# B&R Automation Studio project NAELD004C00R10L518F00 (part 16)

#### Act_OptP0950Ctrl.st
```iecst
ACTION Act_OptP0950Ctrl:

////Control
//	IF g_tyP0950Simu.tySimu.tyHotspotSimu.bRtCompl = TRUE THEN
//		g_tyP0950Simu.tySimu.tyHotspotSimu.bRtCompl	:= FALSE;
//
//		fUIInRtStatOff(ADR(g_tyP0950Simu.tySimuCtrl.tyLyr.uiRtStat));
//	END_IF
//
//	IF g_tyP0950Simu.tySimuCtrl.tyLyr.uiRtStat.0 = FALSE THEN
//		IF g_tyP0950Simu.tySimuCtrl.tyBtnStart.bRtCompl = TRUE THEN
//			g_tyP0950Simu.tySimuCtrl.tyBtnStart.bRtComplm	:= FALSE;
//
//			IF tyOpsProgData.bSimuCycStpCtrl = TRUE THEN
//				tyOpsProgData.bSimuCycStpCtrl	:= FALSE;
//			END_IF
//
//			IF tyOpsProgData.bAutoStepCtrl = TRUE THEN
//				tyOpsProgData.bAutoStepCtrl	:= FALSE;
//			END_IF
//
//			tyOpsProgData.bSimuCtrl	:= TRUE;
//			fUIInRtStatHide(ADR(g_tyP0950Simu.tySimuCtrl.tyLyr.uiRtStat));
//
//		ELSIF g_tyP0950Simu.tySimuCtrl.tyBtnStop.bRtCompl = TRUE THEN
//			g_tyP0950Simu.tySimuCtrl.tyBtnStop.bRtCompl	:= FALSE;
//
//			tyOpsProgData.bSimuCycStpCtrl	:= TRUE;
//			fUIInRtStatHide(ADR(g_tyP0950Simu.tySimuCtrl.tyLyr.uiRtStat));
//
//		ELSIF g_tyP0950Simu.tySimuCtrl.tyBtnStep.bRtCompl = TRUE THEN
//			g_tyP0950Simu.tySimuCtrl.tyBtnStep.bRtCompl	:= FALSE;
//
//			IF tyOpsProgData.bAutoStepCtrl = FALSE THEN
//				tyOpsProgData.bSimuCtrl			:= TRUE;
//				tyOpsProgData.bAutoStepCtrl		:= TRUE;
//				tyOpsProgData.bSimuCycStpCtrl	:= FALSE;
//			ELSIF tyOpsProgData.bSimuCycStpCtrl = TRUE THEN
//				tyOpsProgData.bSimuCycStpCtrl	:= FALSE;
//			ELSE
//				tyOpsProgData.bAutoStepRunCtrl	:= TRUE;
//			END_IF
//		ELSIF g_tyP0950Simu.tySimuCtrl.tyHotspotClose.bRtCompl = TRUE THEN
//			g_tyP0950Simu.tySimuCtrl.tyHotspotClose.bRtCompl	:= FALSE;
//
//			fUIInRtStatHide(ADR(g_tyP0950Simu.tySimuCtrl.tyLyr.uiRtStat));
//		END_IF
//	END_IF
//
//	//Display
//	IF tyOpsProgData.bSimuCtrl = TRUE AND tyOpsProgData.bSimuCycStpCtrl = TRUE THEN
//		fUIInRtStatOff(ADR(g_tyP0950Simu.tySimu.tyBtnStartStat.uiRtStat));
//		fUIInRtStatHide(ADR(g_tyP0950Simu.tySimu.tyBtnStopStat.uiRtStat));
//		fUIInRtStatHide(ADR(g_tyP0950Simu.tySimu.tyBtnStepStat.uiRtStat));
//
//		fbStopBlinkTm(IN := TRUE);
//		IF fbStopBlinkTm.Q = TRUE THEN
//			fbStopBlinkTm(IN := FALSE);
//
//			g_tyP0950Simu.tySimu.tyBtnStartStat.bValue	:= NOT g_tyP0950Simu.tySimu.tyBtnStartStat.bValue;
//		END_IF
//	ELSIF tyOpsProgData.bSimuCtrl = TRUE AND tyOpsProgData.bAutoStepCtrl = TRUE THEN
//		fUIInRtStatHide(ADR(g_tyP0950Simu.tySimu.tyBtnStartStat.uiRtStat));
//		fUIInRtStatHide(ADR(g_tyP0950Simu.tySimu.tyBtnStopStat.uiRtStat));
//		fUIInRtStatOff(ADR(g_tyP0950Simu.tySimu.tyBtnStepStat.uiRtStat));
//	ELSIF tyOpsProgData.bSimuCtrl = TRUE THEN
//		fUIInRtStatOff(ADR(g_tyP0950Simu.tySimu.tyBtnStartStat.uiRtStat));
//		fUIInRtStatHide(ADR(g_tyP0950Simu.tySimu.tyBtnStopStat.uiRtStat));
//		fUIInRtStatHide(ADR(g_tyP0950Simu.tySimu.tyBtnStepStat.uiRtStat));
//
//		g_tyP0950Simu.tySimu.tyBtnStartStat.bValue	:= FALSE;
//	ELSE
//		fUIInRtStatHide(ADR(g_tyP0950Simu.tySimu.tyBtnStartStat.uiRtStat));
//		fUIInRtStatOff(ADR(g_tyP0950Simu.tySimu.tyBtnStopStat.uiRtStat));
//		fUIInRtStatHide(ADR(g_tyP0950Simu.tySimu.tyBtnStepStat.uiRtStat));
//	END_IF
//
//	//Mask
//	IF bErr = TRUE THEN
//		fUIInRtStatOff(ADR(g_tyP0950Simu.tySimu.tyHotspotSimu.uiMaskRtStat));
//	ELSE
//		fUIInRtStatHide(ADR(g_tyP0950Simu.tySimu.tyHotspotSimu.uiMaskRtStat));
//	END_IF

	// Error
	IF EDGEPOS(p_bAlarmErr = TRUE AND p_bSimuStatusStop = FALSE) THEN

		tyP0950Simu.tySimu.tyBtnStart.bRtCompl	:= FALSE;
		tyP0950Simu.tySimu.tyBtnStop.bRtCompl	:= FALSE;
		tyP0950Simu.tySimu.tyBtnInShutterSim.bRtCompl	:= FALSE;

		tyP0950Simu.tySimu.tyBtnStart.bValue	:= FALSE;
		tyP0950Simu.tySimu.tyBtnStop.bValue		:= FALSE;
		tyP0950Simu.tySimu.tyBtnInShutterSim.bValue	:= FALSE;

		eSimuAct	:= SimulationsActError;

	ELSE

		IF p_eSimuStat = SimulationsActError AND p_eSimuStatus = Done THEN
			eSimuAct	:= SimulationsActIdle;

		END_IF

	END_IF

	//Control
	IF tyP0950Simu.tySimu.tyBtnStart.bRtCompl = TRUE THEN
		tyP0950Simu.tySimu.tyBtnStop.bRtCompl	:= FALSE;

		eSimuAct		:= SimulationsActStart;

		IF p_eSimuStat = SimulationsActStart AND p_eSimuStatus = Done THEN
			eSimuAct	:= SimulationsActIdle;

			tyP0950Simu.tySimu.tyBtnStart.bRtCompl	:= FALSE;

		END_IF

	ELSIF tyP0950Simu.tySimu.tyBtnStop.bRtCompl = TRUE THEN
		tyP0950Simu.tySimu.tyBtnStart.bRtCompl	:= FALSE;

		eSimuAct			:= SimulationsActStop;

		IF p_eSimuStat = SimulationsActStop AND p_eSimuStatus = Done THEN
			eSimuAct		:= SimulationsActIdle;

			tyP0950Simu.tySimu.tyBtnStop.bRtCompl	:= FALSE;
		END_IF

	END_IF

	// Mask
	IF p_bAlarmErr = TRUE OR (p_tyDI.bSafetyRlySig = FALSE) THEN
		fUIInRtStatOff(ADR(tyP0950Simu.tySimu.tyBtnStart.uiMaskRtStat));
		fUIInRtStatOff(ADR(tyP0950Simu.tySimu.tyBtnStop.uiMaskRtStat));

	ELSIF p_bSimuStatusCycleStop = TRUE THEN
		fUIInRtStatHide(ADR(tyP0950Simu.tySimu.tyBtnStart.uiMaskRtStat));
		fUIInRtStatOff(ADR(tyP0950Simu.tySimu.tyBtnStop.uiMaskRtStat));

		fbStopBlinkTm(IN := TRUE);
		IF fbStopBlinkTm.Q = TRUE THEN
			fbStopBlinkTm(IN := FALSE);

			tyP0950Simu.tySimu.tyBtnStart.bValue		:= NOT tyP0950Simu.tySimu.tyBtnStart.bValue;
		END_IF

	ELSIF p_bSimuStatusRun = TRUE THEN
		fUIInRtStatOff(ADR(tyP0950Simu.tySimu.tyBtnStart.uiMaskRtStat));
		fUIInRtStatHide(ADR(tyP0950Simu.tySimu.tyBtnStop.uiMaskRtStat));

	ELSE
		fUIInRtStatHide(ADR(tyP0950Simu.tySimu.tyBtnStart.uiMaskRtStat));
		fUIInRtStatOff(ADR(tyP0950Simu.tySimu.tyBtnStop.uiMaskRtStat));

	END_IF

	//AGV Simulatiom
	IF tyP0950Simu.tyAGVToMc.tyBtnAGVSimulateOn.bRtCompl THEN
		IF tyP0950Simu.tyAGVToMc.tyBtnAGVSimulateOn.bValue THEN
			bAGVSimulationOn	:= TRUE;
			tyP0950Simu.tyAGVToMc.tyBtnAGVSimulateOn.bRtCompl:= FALSE;
		ELSE
			bAGVSimulationOn := FALSE;
			tyP0950Simu.tyAGVToMc.tyBtnAGVSimulateOn.bRtCompl:= FALSE;
		END_IF
	END_IF

	IF tyP0950Simu.tyAGVToMc.tyBtnAGVOnline.bRtCompl THEN
		IF tyP0950Simu.tyAGVToMc.tyBtnAGVOnline.bValue THEN
			bAGVSimulateOnline := TRUE;
			tyP0950Simu.tyAGVToMc.tyBtnAGVOnline.bRtCompl := FALSE;
		ELSE
			bAGVSimulateOnline := FALSE;
			tyP0950Simu.tyAGVToMc.tyBtnAGVOnline.bRtCompl := FALSE;
		END_IF
	END_IF

	IF tyP0950Simu.tyAGVToMc.tyBtnAGVAuto.bRtCompl THEN
		IF tyP0950Simu.tyAGVToMc.tyBtnAGVAuto.bValue THEN
			tyAGVSimulateSig.bVEHAuto := TRUE;
			tyP0950Simu.tyAGVToMc.tyBtnAGVAuto.bRtCompl:= FALSE;
		ELSE
			tyAGVSimulateSig.bVEHAuto := FALSE;
			tyP0950Simu.tyAGVToMc.tyBtnAGVAuto.bRtCompl:= FALSE;
		END_IF
	END_IF

	IF tyP0950Simu.tyAGVToMc.tyBtnAGVInPos1.bRtCompl THEN
		IF tyP0950Simu.tyAGVToMc.tyBtnAGVInPos1.bValue THEN
			tyAGVSimulateSig.bVEHInPos1 := TRUE;
			tyP0950Simu.tyAGVToMc.tyBtnAGVInPos1.bRtCompl:= FALSE;
		ELSE
			tyAGVSimulateSig.bVEHInPos1 := FALSE;
			tyP0950Simu.tyAGVToMc.tyBtnAGVInPos1.bRtCompl:= FALSE;
		END_IF
	END_IF

	IF tyP0950Simu.tyAGVToMc.tyBtnAGVInPos2.bRtCompl THEN
		IF tyP0950Simu.tyAGVToMc.tyBtnAGVInPos2.bValue THEN
			tyAGVSimulateSig.bVEHInPos2 := TRUE;
			tyP0950Simu.tyAGVToMc.tyBtnAGVInPos2.bRtCompl:= FALSE;
		ELSE
			tyAGVSimulateSig.bVEHInPos2 := FALSE;
			tyP0950Simu.tyAGVToMc.tyBtnAGVInPos2.bRtCompl:= FALSE;
		END_IF
	END_IF

	IF tyP0950Simu.tyAGVToMc.tyBtnAGVInPos3.bRtCompl THEN
		IF tyP0950Simu.tyAGVToMc.tyBtnAGVInPos3.bValue THEN
			tyAGVSimulateSig.bVEHInPos3 := TRUE;
			tyP0950Simu.tyAGVToMc.tyBtnAGVInPos3.bRtCompl:= FALSE;
		ELSE
			tyAGVSimulateSig.bVEHInPos3 := FALSE;
			tyP0950Simu.tyAGVToMc.tyBtnAGVInPos3.bRtCompl:= FALSE;
		END_IF
	END_IF

	IF tyP0950Simu.tyAGVToMc.tyBtnAGV1Occupied.bRtCompl THEN
		IF tyP0950Simu.tyAGVToMc.tyBtnAGV1Occupied.bValue THEN
			tyAGVSimulateSig.bVEH1Occupied := TRUE;
			tyP0950Simu.tyAGVToMc.tyBtnAGV1Occupied.bRtCompl := FALSE;
		ELSE
			tyAGVSimulateSig.bVEH1Occupied := FALSE;
			tyP0950Simu.tyAGVToMc.tyBtnAGV1Occupied.bRtCompl := FALSE;
		END_IF
	END_IF

	IF tyP0950Simu.tyAGVToMc.tyBtnAGV2Occupied.bRtCompl THEN
		IF tyP0950Simu.tyAGVToMc.tyBtnAGV2Occupied.bValue THEN
			tyAGVSimulateSig.bVEH2Occupied := TRUE;
			tyP0950Simu.tyAGVToMc.tyBtnAGV2Occupied.bRtCompl := FALSE;
		ELSE
			tyAGVSimulateSig.bVEH2Occupied := FALSE;
			tyP0950Simu.tyAGVToMc.tyBtnAGV2Occupied.bRtCompl := FALSE;
		END_IF
	END_IF

	IF tyP0950Simu.tyAGVToMc.tyBtnAGV3Occupied.bRtCompl THEN
		IF tyP0950Simu.tyAGVToMc.tyBtnAGV3Occupied.bValue THEN
			tyAGVSimulateSig.bVEH3Occupied := TRUE;
			tyP0950Simu.tyAGVToMc.tyBtnAGV3Occupied.bRtCompl := FALSE;
		ELSE
			tyAGVSimulateSig.bVEH3Occupied := FALSE;
			tyP0950Simu.tyAGVToMc.tyBtnAGV3Occupied.bRtCompl := FALSE;
		END_IF
	END_IF

	//Machine to AGV Communication
	tyP0950Simu.tyMcToAGV.tyBtnMachineOnline.bValue := p_bMachineOnline;
	tyP0950Simu.tyMcToAGV.tyBtnMachineEstop.bValue	:= p_tyDTMagToAGV.bEStopErr;

	//Magazine #1 to AGV Communication
	tyP0950Simu.tyMcToAGV.tyBtnMag1Auto.bValue				:= p_tyDTMagToAGV.bCI1Auto;
	tyP0950Simu.tyMcToAGV.tyBtnMag1Empty.bValue				:= p_tyDTMagToAGV.bCI1MagazineEmpty;
	tyP0950Simu.tyMcToAGV.tyBtnMag1IncorrectModel.bValue	:= p_tyDTMagToAGV.bCI1IncorrectMagazineModel;
	tyP0950Simu.tyMcToAGV.tyBtnMag1Occupied.bValue			:= p_tyDTMagToAGV.bCI1Occupied;
	tyP0950Simu.tyMcToAGV.tyBtnMag1Rdy.bValue				:= p_tyDTMagToAGV.bCI1Rdy;

	//Magazine #2 to AGV Communication
	tyP0950Simu.tyMcToAGV.tyBtnMag2Auto.bValue				:= p_tyDTMagToAGV.bCI2Auto;
	tyP0950Simu.tyMcToAGV.tyBtnMag2Empty.bValue				:= p_tyDTMagToAGV.bCI2MagazineEmpty;
	tyP0950Simu.tyMcToAGV.tyBtnMag2IncorrectModel.bValue	:= p_tyDTMagToAGV.bCI2IncorrectMagazineModel;
	tyP0950Simu.tyMcToAGV.tyBtnMag2Occupied.bValue			:= p_tyDTMagToAGV.bCI2Occupied;
	tyP0950Simu.tyMcToAGV.tyBtnMag2Rdy.bValue				:= p_tyDTMagToAGV.bCI2Rdy;

	//Magazine #3 to AGV Communication
	tyP0950Simu.tyMcToAGV.tyBtnMag3Auto.bValue				:= p_tyDTMagToAGV.bCI3Auto;
	tyP0950Simu.tyMcToAGV.tyBtnMag3Empty.bValue				:= p_tyDTMagToAGV.bCI3MagazineEmpty;
	tyP0950Simu.tyMcToAGV.tyBtnMag3IncorrectModel.bValue	:= p_tyDTMagToAGV.bCI3IncorrectMagazineModel;
	tyP0950Simu.tyMcToAGV.tyBtnMag3Occupied.bValue			:= p_tyDTMagToAGV.bCI3Occupied;
	tyP0950Simu.tyMcToAGV.tyBtnMag3Rdy.bValue				:= p_tyDTMagToAGV.bCI3Rdy;

	//SOT
	tyP0950Simu.tySimu.tyBtnMagSOT1.tyBtnError.bValue	:= p_tyDO.bSOT1MagError;
	tyP0950Simu.tySimu.tyBtnMagSOT1.tyBtnRdy.bValue		:= p_tyDO.bSOT1MagReady;
	tyP0950Simu.tySimu.tyBtnMagSOT1.tyBtnAvail.bValue	:= p_tyDO.bSOT1MagAvailable;
	tyP0950Simu.tySimu.tyBtnMagSOT1.tyBtnSize.bValue	:= p_tyDO.bSOT1MagSizeLarge;

	tyP0950Simu.tySimu.tyBtnMagSOT2.tyBtnError.bValue	:= p_tyDO.bSOT2MagError;
	tyP0950Simu.tySimu.tyBtnMagSOT2.tyBtnRdy.bValue		:= p_tyDO.bSOT2MagReady;
	tyP0950Simu.tySimu.tyBtnMagSOT2.tyBtnAvail.bValue	:= p_tyDO.bSOT2MagAvailable;
	tyP0950Simu.tySimu.tyBtnMagSOT2.tyBtnSize.bValue	:= p_tyDO.bSOT2MagSizeLarge;

	tyP0950Simu.tySimu.tyBtnMagSOT3.tyBtnError.bValue	:= p_tyDO.bSOT3MagError;
	tyP0950Simu.tySimu.tyBtnMagSOT3.tyBtnRdy.bValue		:= p_tyDO.bSOT3MagReady;
	tyP0950Simu.tySimu.tyBtnMagSOT3.tyBtnAvail.bValue	:= p_tyDO.bSOT3MagAvailable;
	tyP0950Simu.tySimu.tyBtnMagSOT3.tyBtnSize.bValue	:= p_tyDO.bSOT3MagSizeLarge;

	tyP0950Simu.tySimu.tyBtnMagSOT4.tyBtnError.bValue	:= p_tyDO.bSOT4MagError;
	tyP0950Simu.tySimu.tyBtnMagSOT4.tyBtnRdy.bValue		:= p_tyDO.bSOT4MagReady;
	tyP0950Simu.tySimu.tyBtnMagSOT4.tyBtnAvail.bValue	:= p_tyDO.bSOT4MagAvailable;
	tyP0950Simu.tySimu.tyBtnMagSOT4.tyBtnSize.bValue	:= p_tyDO.bSOT4MagSizeLarge;

	//SOT1
	IF tyP0950Simu.tySimu.tyBtnSOT1.tyBtnInPos.bRtCompl THEN
		IF tyP0950Simu.tySimu.tyBtnSOT1.tyBtnInPos.bValue THEN
			tySOTSimulateSig1.tyBtnInPos := TRUE;
			tyP0950Simu.tySimu.tyBtnSOT1.tyBtnInPos.bRtCompl := FALSE;
		ELSE
			tySOTSimulateSig1.tyBtnInPos:= FALSE;
			tyP0950Simu.tySimu.tyBtnSOT1.tyBtnInPos.bRtCompl:= FALSE;
		END_IF
	END_IF

	IF tyP0950Simu.tySimu.tyBtnSOT1.tyBtnRdy.bRtCompl THEN
		IF tyP0950Simu.tySimu.tyBtnSOT1.tyBtnRdy.bValue THEN
			tySOTSimulateSig1.tyBtnRdy := TRUE;
			tyP0950Simu.tySimu.tyBtnSOT1.tyBtnRdy.bRtCompl := FALSE;
		ELSE
			tySOTSimulateSig1.tyBtnRdy := FALSE;
			tyP0950Simu.tySimu.tyBtnSOT1.tyBtnRdy.bRtCompl:= FALSE;
		END_IF
	END_IF

	IF tyP0950Simu.tySimu.tyBtnSOT1.tyBtnAvail.bRtCompl THEN
		IF tyP0950Simu.tySimu.tyBtnSOT1.tyBtnAvail.bValue THEN
			tySOTSimulateSig1.tyBtnAvail := TRUE;
			tyP0950Simu.tySimu.tyBtnSOT1.tyBtnAvail.bRtCompl := FALSE;
		ELSE
			tySOTSimulateSig1.tyBtnAvail:= FALSE;
			tyP0950Simu.tySimu.tyBtnSOT1.tyBtnAvail.bRtCompl:= FALSE;
		END_IF
	END_IF

	IF tyP0950Simu.tySimu.tyBtnSOT1.tyBtnError.bRtCompl THEN
		IF tyP0950Simu.tySimu.tyBtnSOT1.tyBtnError.bValue THEN
			tySOTSimulateSig1.tyBtnError := TRUE;
			tyP0950Simu.tySimu.tyBtnSOT1.tyBtnError.bRtCompl := FALSE;
		ELSE
			tySOTSimulateSig1.tyBtnError:= FALSE;
			tyP0950Simu.tySimu.tyBtnSOT1.tyBtnError.bRtCompl:= FALSE;
		END_IF
	END_IF

	//SOT2
	IF tyP0950Simu.tySimu.tyBtnSOT2.tyBtnInPos.bRtCompl THEN
		IF tyP0950Simu.tySimu.tyBtnSOT2.tyBtnInPos.bValue THEN
			tySOTSimulateSig2.tyBtnInPos := TRUE;
			tyP0950Simu.tySimu.tyBtnSOT2.tyBtnInPos.bRtCompl := FALSE;
		ELSE
			tySOTSimulateSig2.tyBtnInPos:= FALSE;
			tyP0950Simu.tySimu.tyBtnSOT2.tyBtnInPos.bRtCompl:= FALSE;
		END_IF
	END_IF

	IF tyP0950Simu.tySimu.tyBtnSOT2.tyBtnRdy.bRtCompl THEN
		IF tyP0950Simu.tySimu.tyBtnSOT2.tyBtnRdy.bValue THEN
			tySOTSimulateSig2.tyBtnRdy := TRUE;
			tyP0950Simu.tySimu.tyBtnSOT2.tyBtnRdy.bRtCompl := FALSE;
		ELSE
			tySOTSimulateSig2.tyBtnRdy := FALSE;
			tyP0950Simu.tySimu.tyBtnSOT2.tyBtnRdy.bRtCompl:= FALSE;
		END_IF
	END_IF

	IF tyP0950Simu.tySimu.tyBtnSOT2.tyBtnAvail.bRtCompl THEN
		IF tyP0950Simu.tySimu.tyBtnSOT2.tyBtnAvail.bValue THEN
			tySOTSimulateSig2.tyBtnAvail := TRUE;
			tyP0950Simu.tySimu.tyBtnSOT2.tyBtnAvail.bRtCompl := FALSE;
		ELSE
			tySOTSimulateSig2.tyBtnAvail:= FALSE;
			tyP0950Simu.tySimu.tyBtnSOT2.tyBtnAvail.bRtCompl:= FALSE;
		END_IF
	END_IF

	IF tyP0950Simu.tySimu.tyBtnSOT2.tyBtnError.bRtCompl THEN
		IF tyP0950Simu.tySimu.tyBtnSOT2.tyBtnError.bValue THEN
			tySOTSimulateSig2.tyBtnError := TRUE;
			tyP0950Simu.tySimu.tyBtnSOT2.tyBtnError.bRtCompl := FALSE;
		ELSE
			tySOTSimulateSig2.tyBtnError:= FALSE;
			tyP0950Simu.tySimu.tyBtnSOT2.tyBtnError.bRtCompl:= FALSE;
		END_IF
	END_IF

	//SOT3
	IF tyP0950Simu.tySimu.tyBtnSOT3.tyBtnInPos.bRtCompl THEN
		IF tyP0950Simu.tySimu.tyBtnSOT3.tyBtnInPos.bValue THEN
			tySOTSimulateSig3.tyBtnInPos := TRUE;
			tyP0950Simu.tySimu.tyBtnSOT3.tyBtnInPos.bRtCompl := FALSE;
		ELSE
			tySOTSimulateSig3.tyBtnInPos:= FALSE;
			tyP0950Simu.tySimu.tyBtnSOT3.tyBtnInPos.bRtCompl:= FALSE;
		END_IF
	END_IF

	IF tyP0950Simu.tySimu.tyBtnSOT3.tyBtnRdy.bRtCompl THEN
		IF tyP0950Simu.tySimu.tyBtnSOT3.tyBtnRdy.bValue THEN
			tySOTSimulateSig3.tyBtnRdy := TRUE;
			tyP0950Simu.tySimu.tyBtnSOT3.tyBtnRdy.bRtCompl := FALSE;
		ELSE
			tySOTSimulateSig3.tyBtnRdy := FALSE;
			tyP0950Simu.tySimu.tyBtnSOT3.tyBtnRdy.bRtCompl:= FALSE;
		END_IF
	END_IF

	IF tyP0950Simu.tySimu.tyBtnSOT3.tyBtnAvail.bRtCompl THEN
		IF tyP0950Simu.tySimu.tyBtnSOT3.tyBtnAvail.bValue THEN
			tySOTSimulateSig3.tyBtnAvail := TRUE;
			tyP0950Simu.tySimu.tyBtnSOT3.tyBtnAvail.bRtCompl := FALSE;
		ELSE
			tySOTSimulateSig3.tyBtnAvail:= FALSE;
			tyP0950Simu.tySimu.tyBtnSOT3.tyBtnAvail.bRtCompl:= FALSE;
		END_IF
	END_IF

	IF tyP0950Simu.tySimu.tyBtnSOT3.tyBtnError.bRtCompl THEN
		IF tyP0950Simu.tySimu.tyBtnSOT3.tyBtnError.bValue THEN
			tySOTSimulateSig3.tyBtnError := TRUE;
			tyP0950Simu.tySimu.tyBtnSOT3.tyBtnError.bRtCompl := FALSE;
		ELSE
			tySOTSimulateSig3.tyBtnError:= FALSE;
			tyP0950Simu.tySimu.tyBtnSOT3.tyBtnError.bRtCompl:= FALSE;
		END_IF
	END_IF

	//SOT4
	IF tyP0950Simu.tySimu.tyBtnSOT4.tyBtnInPos.bRtCompl THEN
		IF tyP0950Simu.tySimu.tyBtnSOT4.tyBtnInPos.bValue THEN
			tySOTSimulateSig4.tyBtnInPos := TRUE;
			tyP0950Simu.tySimu.tyBtnSOT4.tyBtnInPos.bRtCompl := FALSE;
		ELSE
			tySOTSimulateSig4.tyBtnInPos:= FALSE;
			tyP0950Simu.tySimu.tyBtnSOT4.tyBtnInPos.bRtCompl:= FALSE;
		END_IF
	END_IF

	IF tyP0950Simu.tySimu.tyBtnSOT4.tyBtnRdy.bRtCompl THEN
		IF tyP0950Simu.tySimu.tyBtnSOT4.tyBtnRdy.bValue THEN
			tySOTSimulateSig4.tyBtnRdy := TRUE;
			tyP0950Simu.tySimu.tyBtnSOT4.tyBtnRdy.bRtCompl := FALSE;
		ELSE
			tySOTSimulateSig4.tyBtnRdy := FALSE;
			tyP0950Simu.tySimu.tyBtnSOT4.tyBtnRdy.bRtCompl:= FALSE;
		END_IF
	END_IF
	IF tyP0950Simu.tySimu.tyBtnSOT4.tyBtnAvail.bRtCompl THEN
		IF tyP0950Simu.tySimu.tyBtnSOT4.tyBtnAvail.bValue THEN
			tySOTSimulateSig4.tyBtnAvail := TRUE;
			tyP0950Simu.tySimu.tyBtnSOT4.tyBtnAvail.bRtCompl := FALSE;
		ELSE
			tySOTSimulateSig4.tyBtnAvail:= FALSE;
			tyP0950Simu.tySimu.tyBtnSOT4.tyBtnAvail.bRtCompl:= FALSE;
		END_IF
	END_IF

	IF tyP0950Simu.tySimu.tyBtnSOT4.tyBtnError.bRtCompl THEN
		IF tyP0950Simu.tySimu.tyBtnSOT4.tyBtnError.bValue THEN
			tySOTSimulateSig4.tyBtnError := TRUE;
			tyP0950Simu.tySimu.tyBtnSOT4.tyBtnError.bRtCompl := FALSE;
		ELSE
			tySOTSimulateSig4.tyBtnError:= FALSE;
			tyP0950Simu.tySimu.tyBtnSOT4.tyBtnError.bRtCompl:= FALSE;
		END_IF
	END_IF

	//InShutter Sim
	IF tyP0950Simu.tySimu.tyBtnInShutterSim.bValue THEN
		usiSimuMod := 1;// shutter sim
		IF fbShutterSimChgOver.Q OR tyP0950Simu.tySimu.tyBtnInShutterSim.bRtCompl THEN
			tyP0950Simu.tySimu.tyBtnInShutterSim.bRtCompl := FALSE;
			fbShutterSimChgOver (IN:= FALSE);
			IF p_tyDI.bInShutterCloseRS AND (p_tyDI.bInShutterCloseRS2 OR p_tyNtParamCurr.bProjShutter2Prep = FALSE) AND
				(p_tyDI.bInShutterCloseRS3 OR p_tyNtParamCurr.bProjShutter3Prep = FALSE) AND p_tyDI.bOutShutterCloseRS THEN
				eInShutterAct  := PneuActRet;
				eInShutterAct2 := PneuActRet;
				eInShutterAct3 := PneuActRet;
				eOutShutterAct := PneuActRet;
			ELSIF p_tyDI.bInShutterOpenRS AND (p_tyDI.bInShutterOpenRS2 OR p_tyNtParamCurr.bProjShutter2Prep = FALSE) AND
				(p_tyDI.bInShutterOpenRS3 OR p_tyNtParamCurr.bProjShutter3Prep = FALSE)AND p_tyDI.bOutShutterOpenRS THEN
				eInShutterAct  := PneuActExt;
				eInShutterAct2 := PneuActExt;
				eInShutterAct3 := PneuActExt;
				eOutShutterAct := PneuActExt;
			END_IF
		ELSIF fbShutterSimChgOver.ET = T#5s THEN

		END_IF

		IF p_eInShutterStatus = Done AND (p_eInShutterStatus2 = Done OR p_tyNtParamCurr.bProjShutter2Prep = FALSE) AND
			(p_eInShutterStatus3 = Done OR p_tyNtParamCurr.bProjShutter3Prep = FALSE) AND p_eOutShutterStatus = Done THEN
			eInShutterAct  := PneuActIdle;
			eInShutterAct2 := PneuActIdle;
			eInShutterAct3 := PneuActIdle;
			eOutShutterAct := PneuActIdle;
			fbShutterSimChgOver (IN:= TRUE);
		END_IF
		fbShutterSimChgOver;
	ELSE
		eInShutterAct  := PneuActIdle;
		eInShutterAct2 := PneuActIdle;
		eInShutterAct3 := PneuActIdle;
		eOutShutterAct := PneuActIdle;

	END_IF

	//Test trav
	IF tyP0950Simu.tySimu.tyBtnTestTrav.bValue THEN
		CASE usiTestTravStep OF
			0:
				eTravAct		:= TravActGoAPos;

				IF p_eTravStat = TravActGoAPos AND p_eTravStatus = Done THEN
					eTravAct	:= TravActIdle;
					usiTestTravStep := 1;
				END_IF
			1:

				eTravAct		:= TravActGoCPos;

				IF p_eTravStat = TravActGoCPos AND p_eTravStatus = Done THEN
					eTravAct	:= TravActIdle;
					usiTestTravStep := 0;
				END_IF
		END_CASE
		diMnlTravNomSpd		:= 1500000;
	ELSE
		eTravAct		:= TravActIdle;
		diMnlTravNomSpd		:= 0;
	END_IF

	//NT- speed
	IF tyP0950Simu.tySimu.tyBtnNtParaWr2.bValue AND usiSimuMod =1 AND usiSimuNtStep = 0 THEN
		eTravAct		:= TravActIdle;
		p_diNtParamTravAutoSpd 		:= tyP0950Simu.tySimu.tyNumTravSpd.diValue;
		p_diNtParamLifterAutoSpd	:= tyP0950Simu.tySimu.tyNumLifterSpd.diValue;
		eNtWr := 3;
		IF p_eNtParamStat = 3 AND p_eNtParamStatus = Done THEN
			CASE usiWrStep OF
				0:

					memcpy(ADR(fbSDOWriteAccT.data0),ADR(udiAcc),1);
					memcpy(ADR(fbSDOWriteAccT.data1),ADR(udiAcc)+1,1);
					memcpy(ADR(fbSDOWriteAccL.data0),ADR(udiAcc),1);
					memcpy(ADR(fbSDOWriteAccL.data1),ADR(udiAcc)+1,1);
					fbSDOWriteAccT(enable := TRUE,index := 16#6083, subindex := 0, datalen := 4);
					fbSDOWriteAccL(enable := TRUE,index := 16#6083, subindex := 0, datalen := 4);
					IF fbSDOWriteAccT.status = 65535 AND fbSDOWriteAccL.status = 65535 THEN
						usiWrStep := 1;
					END_IF

				1:
					fbSDOWriteAccT(enable := TRUE);
					fbSDOWriteAccL(enable := TRUE);
					IF fbSDOWriteAccT.status = 0 AND fbSDOWriteAccL.status = 0 THEN
						fbSDOWriteAccT(enable := FALSE);
						fbSDOWriteAccL(enable := FALSE);
						usiWrStep := 2;
//						tyP0950Simu.tySimu.tyBtnNtParaWr2.bValue := FALSE;
//						eNtWr := 0;
					END_IF
				2:
					memcpy(ADR(fbSDOWriteAccT.data0),ADR(udiAcc),1);
					memcpy(ADR(fbSDOWriteAccT.data1),ADR(udiAcc)+1,1);
					memcpy(ADR(fbSDOWriteAccL.data0),ADR(udiAcc),1);
					memcpy(ADR(fbSDOWriteAccL.data1),ADR(udiAcc)+1,1);
					fbSDOWriteAccT(enable := TRUE,index := 16#6084, subindex := 0, datalen := 4);
					fbSDOWriteAccL(enable := TRUE,index := 16#6084, subindex := 0, datalen := 4);
					IF fbSDOWriteAccT.status = 65535 AND fbSDOWriteAccL.status = 65535 THEN
						usiWrStep := 3;
					END_IF
				3:
					fbSDOWriteAccT(enable := TRUE);
					fbSDOWriteAccL(enable := TRUE);
					IF fbSDOWriteAccT.status = 0 AND fbSDOWriteAccL.status = 0 THEN
						fbSDOWriteAccT(enable := FALSE);
						fbSDOWriteAccL(enable := FALSE);
						usiWrStep := 0;
						tyP0950Simu.tySimu.tyBtnNtParaWr2.bValue := FALSE;
						eNtWr := 0;
					END_IF

			END_CASE
		END_IF
	END_IF

	//NT -addr and jobno
	IF tyP0950Simu.tySimu.tyBtnNtParaWr.bValue AND usiSimuMod =1 THEN
		p_sNtParamJobNo 		:= tyP0950Simu.tySimu.tyStringJobNo.sValue;
		p_usiNtParamNtAddr 		:= DINT_TO_USINT( tyP0950Simu.tySimu.tyNumAddr.diValue);
		CASE usiSimuNtStep OF
			0:
				eNtWr := 3;
				IF p_eNtParamStat = 3 AND p_eNtParamStatus = Done THEN
					eNtWr := 0;
					usiSimuNtStep := 1;
				END_IF
			1:
				IF  p_eNtParamStatus = Idle THEN
					eNtWr := 5;
				END_IF
				IF p_eNtParamStat = 5 AND p_eNtParamStatus = Done THEN
					eNtWr := 0;
					usiSimuNtStep := 2;
				END_IF
			2:
				p_eAct := 1; //refresh page
				IF eUIInit = UIInitialDone THEN
					p_eAct := 0;
					usiSimuNtStep := 0;
					tyP0950Simu.tySimu.tyBtnNtParaWr.bValue := FALSE;
				END_IF
		END_CASE

	ELSIF usiSimuMod =0 THEN //when reset
		tyP0950Simu.tySimu.tyBtnNtParaWr.bValue := FALSE;
	END_IF

	Act_OptP0950RcpGen;

END_ACTION
```

#### Act_OptP0950RcpGen.st
```iecst
ACTION Act_OptP0950RcpGen:
	//Generate test rcp
	IF tyP0950Simu.tySimu.tyBtnRcpGen.bValue THEN
		p_tyProdRcpCurrList[1].sRcpNm		:= '1';
		p_tyProdRcpCurrList[1].diWidthInUM	:= 100000;
		//		p_tyProdRcpCurrList[1].diWidthInUM2
		p_tyProdRcpCurrList[1].diMaxSltValue := p_tyNtParamCurr.tyProdRcpMaxSlt.diMax;
		p_tyProdRcpCurrList[1].diMinSltValue := p_tyNtParamCurr.tyProdRcpMaxSlt.diMin;
		p_tyProdRcpCurrList[1].diPitch		 := 4;
		//		p_tyProdRcpCurrList[1].usiMcMod
		//		p_tyProdRcpCurrList[1].usiFlippedBrd
		p_tyProdRcpCurrList[1].bTopToBtm	:= p_tyNtParamCurr.bProjTopToBtmDefault;
		//		p_tyProdRcpCurrList[1].bLongBrd

		//		p_tyProdRcpCurrList[1].diWidthInUMRear
		//		p_tyProdRcpCurrList[1].diMaxSltValueRear
		//		p_tyProdRcpCurrList[1].diMinSltValueRear
		//		p_tyProdRcpCurrList[1].diPitchRear
		p_tyProdRcpCurrList[1].diMtrPshrExtSpd 	:= 7;
		p_tyProdRcpCurrList[1].diMtrPshrExtTorq := 80;
		p_tyProdRcpCurrList[1].diPshrOffset		:= 0;
		p_tyProdRcpCurrList[1].sDisplayInfo		:= '100.0mm';

		p_tyProdRcpCurrList[2].sRcpNm		:= '2';
		p_tyProdRcpCurrList[2].diWidthInUM	:= 200000;
		p_tyProdRcpCurrList[2].diMaxSltValue := p_tyNtParamCurr.tyProdRcpMaxSlt.diMax;
		p_tyProdRcpCurrList[2].diMinSltValue := p_tyNtParamCurr.tyProdRcpMaxSlt.diMin;
		p_tyProdRcpCurrList[2].diPitch		 := 2;
		p_tyProdRcpCurrList[2].bTopToBtm	:= p_tyNtParamCurr.bProjTopToBtmDefault;

		p_tyProdRcpCurrList[2].diMtrPshrExtSpd 	:= 7;
		p_tyProdRcpCurrList[2].diMtrPshrExtTorq := 80;
		p_tyProdRcpCurrList[2].diPshrOffset		:= 0;
		p_tyProdRcpCurrList[2].sDisplayInfo		:= '200.0mm';

		p_tyProdRcpCurrList[3].sRcpNm		:= '3';
		p_tyProdRcpCurrList[3].diWidthInUM	:= 250000;
		p_tyProdRcpCurrList[3].diMaxSltValue := p_tyNtParamCurr.tyProdRcpMaxSlt.diMax;
		p_tyProdRcpCurrList[3].diMinSltValue := p_tyNtParamCurr.tyProdRcpMaxSlt.diMin;
		p_tyProdRcpCurrList[3].diPitch		 := 1;
		p_tyProdRcpCurrList[3].bTopToBtm	:= p_tyNtParamCurr.bProjTopToBtmDefault;

		p_tyProdRcpCurrList[3].diMtrPshrExtSpd 	:= 7;
		p_tyProdRcpCurrList[3].diMtrPshrExtTorq := 80;
		p_tyProdRcpCurrList[3].diPshrOffset		:= 0;
		p_tyProdRcpCurrList[3].sDisplayInfo		:= '250.0mm';

		p_tyProdRcpCurrList[4].sRcpNm		:= 'min';
		p_tyProdRcpCurrList[4].diWidthInUM	:= p_tyNtParamCurr.tyProdRcpWidth.diMin;
		p_tyProdRcpCurrList[4].diMaxSltValue := p_tyNtParamCurr.tyProdRcpMaxSlt.diMax;
		p_tyProdRcpCurrList[4].diMinSltValue := p_tyNtParamCurr.tyProdRcpMaxSlt.diMin;
		p_tyProdRcpCurrList[4].diPitch		 := 1;
		p_tyProdRcpCurrList[4].bTopToBtm	:= p_tyNtParamCurr.bProjTopToBtmDefault;

		p_tyProdRcpCurrList[4].diMtrPshrExtSpd 	:= 7;
		p_tyProdRcpCurrList[4].diMtrPshrExtTorq := 80;
		p_tyProdRcpCurrList[4].diPshrOffset		:= 0;
		string1 := DINT_TO_STRING(p_tyNtParamCurr.tyProdRcpWidth.diMin);
		string1 := LEFT(string1,LEN(string1)-3);
		p_tyProdRcpCurrList[4].sDisplayInfo		:= CONCAT(string1,'.0mm');

		p_tyProdRcpCurrList[5].sRcpNm		:= 'max';
		p_tyProdRcpCurrList[5].diWidthInUM	:= p_tyNtParamCurr.tyProdRcpWidth.diMax;
		p_tyProdRcpCurrList[5].diMaxSltValue := p_tyNtParamCurr.tyProdRcpMaxSlt.diMax;
		p_tyProdRcpCurrList[5].diMinSltValue := p_tyNtParamCurr.tyProdRcpMaxSlt.diMin;
		p_tyProdRcpCurrList[5].diPitch		 := 1;
		p_tyProdRcpCurrList[5].bTopToBtm	:= p_tyNtParamCurr.bProjTopToBtmDefault;

		p_tyProdRcpCurrList[5].diMtrPshrExtSpd 	:= 7;
		p_tyProdRcpCurrList[5].diMtrPshrExtTorq := 80;
		p_tyProdRcpCurrList[5].diPshrOffset		:= 0;
		string1 := DINT_TO_STRING(p_tyNtParamCurr.tyProdRcpWidth.diMax);
		string1 := LEFT(string1,LEN(string1)-3);
		p_tyProdRcpCurrList[5].sDisplayInfo		:= CONCAT(string1,'.0mm');

		eProdRcpAct	:= 12; //ProdRcpActSaveList

		IF p_eProdRcpStat = 12 AND p_eProdRcpStatus = Done THEN
			eProdRcpAct	:= ProdRcpActIdle;
			tyP0950Simu.tySimu.tyBtnRcpGen.bValue := FALSE;
		END_IF

	ELSIF p_eProdRcpStatus = Error THEN
		tyP0950Simu.tySimu.tyBtnRcpGen.bValue := FALSE;
	END_IF

END_ACTION
```

#### Act_OptP0950RstMnl.st
```iecst
ACTION Act_OptP0950RstMnl:

	IF eCurrPage <> UIP0950Simu THEN
		usiSimuMod := 0;
		tyP0950Simu.tySimu.tyBtnInShutterSim.bValue := FALSE;

		bAGVSimulationOn := FALSE;
		tyP0950Simu.tyAGVToMc.tyBtnAGVSimulateOn.bValue := FALSE;

		bAGVSimulateOnline := FALSE;
		tyP0950Simu.tyAGVToMc.tyBtnAGVOnline.bValue := FALSE;

		tyAGVSimulateSig.bVEHAuto := FALSE;
		tyP0950Simu.tyAGVToMc.tyBtnAGVAuto.bValue := FALSE;

		tyAGVSimulateSig.bVEH1Occupied := FALSE;
		tyP0950Simu.tyAGVToMc.tyBtnAGV1Occupied.bValue := FALSE;

		tyAGVSimulateSig.bVEH2Occupied := FALSE;
		tyP0950Simu.tyAGVToMc.tyBtnAGV2Occupied.bValue := FALSE;

		tyAGVSimulateSig.bVEH3Occupied := FALSE;
		tyP0950Simu.tyAGVToMc.tyBtnAGV3Occupied.bValue := FALSE;

		tyAGVSimulateSig.bVEHInPos1 := FALSE;
		tyP0950Simu.tyAGVToMc.tyBtnAGVInPos1.bValue := FALSE;

		tyAGVSimulateSig.bVEHInPos2 := FALSE;
		tyP0950Simu.tyAGVToMc.tyBtnAGVInPos2.bValue := FALSE;

		tyAGVSimulateSig.bVEHInPos3 := FALSE;
		tyP0950Simu.tyAGVToMc.tyBtnAGVInPos3.bValue := FALSE;

	END_IF

END_ACTION
```

#### Act_EntP1000Disp.st
```iecst
ACTION Act_EntP1000Disp:

	//Access Address
	p_tyC0005Main ACCESS ADR(tyCommon.tyMain);

	p_tyC0007Notif ACCESS ADR(tyCommon.tyNotif);

	p_tyC0008MsgBox ACCESS ADR(tyP1000Lang.tyMsgBoxHide);

	p_tyC0009Info ACCESS ADR(tyCommon.tyInfo);

	p_tyP1000Lang ACCESS ADR(tyP1000Lang.tyLang);

	//Backup Param
	tyP1000Lang.tyLangBkUp	:= tyP1000Lang.tyLang;

	//Display
	tyP1000Lang.tyLang.tyBtnEnglish.uiRtStat.0			:= NOT (p_tyNtParamCurr.bchineseprep OR p_tyNtParamCurr.bgermanprep);
	tyP1000Lang.tyLang.tyBtnChinese.uiRtStat.0			:= NOT (p_tyNtParamCurr.bchineseprep);
	tyP1000Lang.tyLang.tyBtnGerman.uiRtStat.0			:= NOT (p_tyNtParamCurr.bgermanprep);

END_ACTION
```

#### Act_EntP1020Disp.st
```iecst
ACTION Act_EntP1020Disp:

	//Access Address
	p_tyC0005Main ACCESS ADR(tyCommon.tyMain);

	p_tyC0007Notif ACCESS ADR(tyCommon.tyNotif);

	p_tyC0008MsgBox ACCESS ADR(tyP1020McSetNavi.tyMsgBoxHide);

	p_tyC0009Info ACCESS ADR(tyCommon.tyInfo);

	p_tyP1020McSetNavi ACCESS ADR(tyP1020McSetNavi.tyNavi);

	tyP1020McSetNavi.tyNavi.tyBtnUSBSet.uiRtStat.0 := NOT(p_tyMcParamCurr.bScannerEn AND p_tyNtParamCurr.bUSBScannerPrep);

	//Display
	//new for Hermes 1.3
	IF (p_tyNtParamCurr.bHermesSvyPrep AND p_tyMcParamCurr.bHermesSvyEn)
		OR p_tyNtParamCurr.bLFPrep OR p_tyNtParamCurr.bLCSLFPrep OR p_tyNtParamCurr.bLCSReqRcpPrep OR p_tyNtParamCurr.bLCSLiveDatPrep
		OR p_tyNtParamCurr.bLCSManageRcpPrep OR p_tyNtParamCurr.bLFUsrSetPrep OR p_tyNtParamCurr.bLFUsrSetPrep
		(*OR p_tyNtParamCurr.bUSWidthChkPrep*) OR p_tyNtParamCurr.bDSWidthChkPrep THEN

		fUIInRtStatOff(ADR(tyP1020McSetNavi.tyNavi.tyBtnVCommSet.uiRtStat));
	ELSE
		fUIInRtStatHide(ADR(tyP1020McSetNavi.tyNavi.tyBtnVCommSet.uiRtStat));
	END_IF
END_ACTION
```

#### Act_OptP1020Navi.st
```iecst
ACTION Act_OptP1020Navi:

	IF tyP1020McSetNavi.tyNavi.tyBtnMcSet.bRtCompl = TRUE THEN
		tyP1020McSetNavi.tyNavi.tyBtnMcSet.bRtCompl			:= FALSE;
		tyP1020McSetNavi.tyNavi.tyBtnMcSet.bValue			:= FALSE;

		eChgPage	:= UIP1021McSetGen;

	ELSIF tyP1020McSetNavi.tyNavi.tyBtnVCommSet.bRtCompl = TRUE THEN
		tyP1020McSetNavi.tyNavi.tyBtnVCommSet.bRtCompl		:= FALSE;
		tyP1020McSetNavi.tyNavi.tyBtnVCommSet.bValue		:= FALSE;

		eChgPage	:= UIP1022McSetVComm;

	ELSIF tyP1020McSetNavi.tyNavi.tyBtnHCommSet.bRtCompl = TRUE THEN
		tyP1020McSetNavi.tyNavi.tyBtnHCommSet.bRtCompl		:= FALSE;
		tyP1020McSetNavi.tyNavi.tyBtnHCommSet.bValue		:= FALSE;

		eChgPage	:= UIP1023McSetHComm;

	ELSIF tyP1020McSetNavi.tyNavi.tyBtnAntiGapSet.bRtCompl = TRUE THEN
		tyP1020McSetNavi.tyNavi.tyBtnAntiGapSet.bRtCompl	:= FALSE;
		tyP1020McSetNavi.tyNavi.tyBtnAntiGapSet.bValue		:= FALSE;

		eChgPage	:= UIP1024McSetAntiGap;

	ELSIF tyP1020McSetNavi.tyNavi.tyBtnAIVCommSet.bRtCompl = TRUE THEN
		tyP1020McSetNavi.tyNavi.tyBtnAIVCommSet.bRtCompl	:= FALSE;
		tyP1020McSetNavi.tyNavi.tyBtnAIVCommSet.bValue		:= FALSE;

		eChgPage	:= UIP1025McSetAIVComm;

	ELSIF tyP1020McSetNavi.tyNavi.tyBtnUSBSet.bRtCompl = TRUE THEN
		tyP1020McSetNavi.tyNavi.tyBtnUSBSet.bRtCompl	:= FALSE;
		tyP1020McSetNavi.tyNavi.tyBtnUSBSet.bValue	:= FALSE;

		eChgPage	:= UIP1027McSetUSBSet;

	ELSIF tyP1020McSetNavi.tyNavi.tyBtnRS232Set.bRtCompl = TRUE THEN
		tyP1020McSetNavi.tyNavi.tyBtnRS232Set.bRtCompl	:= FALSE;
		tyP1020McSetNavi.tyNavi.tyBtnRS232Set.bValue	:= FALSE;

		eChgPage	:= UIP1028McSetRS232Set;
	END_IF

END_ACTION
```

#### Act_EntP1021Disp.st
```iecst
ACTION Act_EntP1021Disp:

	//Access Address
	IF bTeachTravPosA OR bTeachTravPosB OR bTeachLifterPosA OR bTeachLifterPosB THEN
		p_tyC0004Navi ACCESS ADR(tyP1021McSetGen.tyNaviLyr2);
		IF p_tyNtParamCurr.tyDISettings.diMagWidthChkSen > 0 THEN
			tyP1021McSetGen.tyNaviLyr2.tyBitmapPageDisp.usiValueIdx := 4;
		ELSE
			tyP1021McSetGen.tyNaviLyr2.tyBitmapPageDisp.usiValueIdx := 2;
		END_IF
	ELSIF p_tyNtParamCurr.tyDISettings.diMagWidthChkSen > 0 THEN
		p_tyC0004Navi ACCESS ADR(tyP1021McSetGen.tyNaviLyr3); //3 lyr
	ELSE
		p_tyC0004Navi ACCESS ADR(tyP1021McSetGen.tyNaviLyr1);
	END_IF

	p_tyC0005Main ACCESS ADR(tyCommon.tyMain);

	p_tyC0006Set ACCESS ADR(tyCommon.tySet);

	p_tyC0007Notif ACCESS ADR(tyCommon.tyNotif);

	p_tyC0008MsgBox ACCESS ADR(tyP1021McSetGen.tyMsgBoxHide);

	p_tyC0009Info ACCESS ADR(tyCommon.tyInfo);

	p_tyP1021McSetGen ACCESS ADR(tyP1021McSetGen.tyGen);

	p_tyP1021McSetNetwork ACCESS ADR(tyP1021McSetGen.tyNetwork);

	//Display
	tyP1021McSetGen.tyGen.tyLyrGen1.uiRtStat.0	:= bTeachTravPosA OR bTeachTravPosB OR bTeachLifterPosA OR bTeachLifterPosB;
	tyP1021McSetGen.tyGen.tyLyrGen2.uiRtStat.0	:= NOT(bTeachTravPosA OR bTeachTravPosB OR bTeachLifterPosA OR bTeachLifterPosB);
	tyP1021McSetGen.tyGen.tyLyrGen3.uiRtStat.0	:= TRUE;//NOT (p_tyNtParamCurr.tyDISettings.diMagWidthChkSen > 0) ;

	//Backup Param
	IF NOT(bTeachTravPosA OR bTeachTravPosB OR bTeachLifterPosA OR bTeachLifterPosB) THEN
		tyP1021McSetGen.tyGenBkUp	:= tyP1021McSetGen.tyGen;
	ELSE
		bTeachTravPosA		:= FALSE;
		bTeachTravPosB		:= FALSE;
		bTeachLifterPosA	:= FALSE;
		bTeachLifterPosB	:= FALSE;
	END_IF

	//Network Configuration Display
	usiNetworkModeOld := DINT_TO_USINT(p_tyMcParamCurr.eNetworkMod);

	fUIInRtStatHide(ADR(tyP1021McSetGen.tyNetwork.tyLyr.uiRtStat));
	bTeachServo					:= FALSE;

	tyP1021McSetGen.tyGen.tyBtnLFBuzMute.uiRtStat.0 := NOT (p_tyMcParamCurr.bLFEn AND p_tyNtParamCurr.bLFPrep AND p_tyNtParamCurr.tyDOSettings.diBuzzer > 0);

	//Outlet Shutter disable //mask when not Siemens with admin
	IF p_tyNtParamCurr.eCustomerReq = Siemens AND p_tyUsrMgmtCurrUsr.eUsrLvl <> UsrMgmtAdmin THEN
		tyP1021McSetGen.tyGen.tyBtnOutShutterDis.uiMaskRtStat := FALSE;
	ELSE
		tyP1021McSetGen.tyGen.tyBtnOutShutterDis.uiMaskRtStat := TRUE; // operation will initial open when dis.
	END_IF

	tyP1021McSetGen.tyGen.tyBtnRFIDEn.bValue := p_tyMcParamCurr.bMesRFIDEn;
	tyP1021McSetGen.tyGen.tyBtnHermesSvyEn.bValue := p_tyMcParamCurr.bHermesSvyEn;
END_ACTION
```

#### Act_ExitP1021.st
```iecst
ACTION Act_ExitP1021:

	IF (tyCommon.tySet.tyBtnSave.uiMaskRtStat.0 = FALSE) OR (bTeachTravPosA OR bTeachTravPosB OR bTeachLifterPosA OR bTeachLifterPosB) THEN
		usiChgPage	:= 1;

	ELSE

		p_tyC0008MsgBox ACCESS ADR(tyP1021McSetGen.tyMsgBoxExitAsk);

		IF tyP1021McSetGen.tyMsgBoxExitAsk.tyBtnYes.bRtCompl = TRUE THEN
			tyP1021McSetGen.tyMsgBoxExitAsk.tyBtnYes.bRtCompl	:= FALSE;
			tyP1021McSetGen.tyMsgBoxExitAsk.tyBtnYes.bValue		:= FALSE;

			p_tyC0008MsgBox ACCESS ADR(tyP1021McSetGen.tyMsgBoxHide);

			//Restore Param
			tyP1021McSetGen.tyGen	:= tyP1021McSetGen.tyGenBkUp;

			fUIInRtStatOff(ADR(tyCommon.tySet.tyBtnSave.uiMaskRtStat));

			bSaveNetworkPriority	:= FALSE;

			usiChgPage	:= 1;

		ELSIF tyP1021McSetGen.tyMsgBoxExitAsk.tyBtnNo.bRtCompl = TRUE THEN
			tyP1021McSetGen.tyMsgBoxExitAsk.tyBtnNo.bRtCompl	:= FALSE;
			tyP1021McSetGen.tyMsgBoxExitAsk.tyBtnNo.bValue		:= FALSE;

			p_tyC0008MsgBox ACCESS ADR(tyP1021McSetGen.tyMsgBoxHide);

			eChgPage	:= eCurrPage;
			usiChgPage	:= 0;

		END_IF

	END_IF

END_ACTION
```

#### Act_OptP1021Navi.st
```iecst
ACTION Act_OptP1021Navi:

	tyP1021McSetGen.tyNaviLyr1.tyBtnBack.bRtLk	:= tyCommon.tySet.tyBtnSave.bRtCompl;
	tyP1021McSetGen.tyNaviLyr2.tyBtnBack.bRtLk	:= tyCommon.tySet.tyBtnSave.bRtCompl;
	tyP1021McSetGen.tyNaviLyr3.tyBtnBack.bRtLk	:= tyCommon.tySet.tyBtnSave.bRtCompl;

	IF tyP1021McSetGen.tyNaviLyr1.tyBtnBack.bRtCompl = TRUE OR tyP1021McSetGen.tyNaviLyr2.tyBtnBack.bRtCompl = TRUE  OR tyP1021McSetGen.tyNaviLyr3.tyBtnBack.bRtCompl THEN
		tyP1021McSetGen.tyNaviLyr1.tyBtnBack.bRtCompl		:= FALSE;
		tyP1021McSetGen.tyNaviLyr2.tyBtnBack.bRtCompl		:= FALSE;
		tyP1021McSetGen.tyNaviLyr3.tyBtnBack.bRtCompl 		:= FALSE;

		eChgPage	:= UIP1020McSetNavi;

	//Navi From Layer 1 to Layer 2
	ELSIF tyP1021McSetGen.tyNaviLyr1.tyBtnRgt.bRtCompl = TRUE THEN
		p_tyC0004Navi ACCESS ADR (tyP1021McSetGen.tyNaviLyr2);
		IF p_tyNtParamCurr.tyDISettings.diMagWidthChkSen > 0 THEN
			tyP1021McSetGen.tyNaviLyr2.tyBitmapPageDisp.usiValueIdx := 4;
		ELSE
			tyP1021McSetGen.tyNaviLyr2.tyBitmapPageDisp.usiValueIdx := 2;
		END_IF

		fUIInRtStatHide(ADR(tyP1021McSetGen.tyGen.tyLyrGen1.uiRtStat));
		fUIInRtStatOff(ADR(tyP1021McSetGen.tyGen.tyLyrGen2.uiRtStat));
		fUIInRtStatHide(ADR(tyP1021McSetGen.tyGen.tyLyrGen3.uiRtStat));

		tyP1021McSetGen.tyNaviLyr1.tyBtnRgt.bRtCompl			:= FALSE;

	ELSIF tyP1021McSetGen.tyNaviLyr1.tyBtnLeft.bRtCompl = TRUE THEN
		IF p_tyNtParamCurr.tyDISettings.diMagWidthChkSen > 0 THEN
			p_tyC0004Navi ACCESS ADR(tyP1021McSetGen.tyNaviLyr3);
			tyP1021McSetGen.tyNaviLyr3.tyBitmapPageDisp.usiValueIdx := 5; //page3
			fUIInRtStatHide(ADR(tyP1021McSetGen.tyGen.tyLyrGen1.uiRtStat));
			fUIInRtStatHide(ADR(tyP1021McSetGen.tyGen.tyLyrGen2.uiRtStat));
			fUIInRtStatOff(ADR(tyP1021McSetGen.tyGen.tyLyrGen3.uiRtStat));
		ELSE
			p_tyC0004Navi ACCESS ADR (tyP1021McSetGen.tyNaviLyr2);

			fUIInRtStatHide(ADR(tyP1021McSetGen.tyGen.tyLyrGen1.uiRtStat));
			fUIInRtStatOff(ADR(tyP1021McSetGen.tyGen.tyLyrGen2.uiRtStat));
			fUIInRtStatHide(ADR(tyP1021McSetGen.tyGen.tyLyrGen3.uiRtStat));
		END_IF

		tyP1021McSetGen.tyNaviLyr1.tyBtnLeft.bRtCompl			:= FALSE;

	//Navi Form Layer 2 to Layer 1
	ELSIF tyP1021McSetGen.tyNaviLyr2.tyBtnRgt.bRtCompl = TRUE THEN
		IF p_tyNtParamCurr.tyDISettings.diMagWidthChkSen > 0 THEN
			p_tyC0004Navi ACCESS ADR(tyP1021McSetGen.tyNaviLyr3);
			tyP1021McSetGen.tyNaviLyr3.tyBitmapPageDisp.usiValueIdx := 5; //page3
			fUIInRtStatHide(ADR(tyP1021McSetGen.tyGen.tyLyrGen1.uiRtStat));
			fUIInRtStatHide(ADR(tyP1021McSetGen.tyGen.tyLyrGen2.uiRtStat));
			fUIInRtStatOff(ADR(tyP1021McSetGen.tyGen.tyLyrGen3.uiRtStat));
		ELSE
			p_tyC0004Navi ACCESS ADR(tyP1021McSetGen.tyNaviLyr1);

			fUIInRtStatOff(ADR(tyP1021McSetGen.tyGen.tyLyrGen1.uiRtStat));
			fUIInRtStatHide(ADR(tyP1021McSetGen.tyGen.tyLyrGen2.uiRtStat));
			fUIInRtStatHide(ADR(tyP1021McSetGen.tyGen.tyLyrGen3.uiRtStat));
		END_IF

		tyP1021McSetGen.tyNaviLyr2.tyBtnRgt.bRtCompl			:= FALSE;

	ELSIF tyP1021McSetGen.tyNaviLyr2.tyBtnLeft.bRtCompl = TRUE THEN
		p_tyC0004Navi ACCESS ADR(tyP1021McSetGen.tyNaviLyr1);
		IF p_tyNtParamCurr.tyDISettings.diMagWidthChkSen > 0 THEN
			tyP1021McSetGen.tyNaviLyr1.tyBitmapPageDisp.usiValueIdx := 3;
		ELSE
			tyP1021McSetGen.tyNaviLyr1.tyBitmapPageDisp.usiValueIdx := 1;
		END_IF

		fUIInRtStatOff(ADR(tyP1021McSetGen.tyGen.tyLyrGen1.uiRtStat));
		fUIInRtStatHide(ADR(tyP1021McSetGen.tyGen.tyLyrGen2.uiRtStat));
		fUIInRtStatHide(ADR(tyP1021McSetGen.tyGen.tyLyrGen3.uiRtStat));

		tyP1021McSetGen.tyNaviLyr2.tyBtnLeft.bRtCompl			:= FALSE;

		//layer 3
	ELSIF  tyP1021McSetGen.tyNaviLyr3.tyBtnRgt.bRtCompl = TRUE THEN
		p_tyC0004Navi ACCESS ADR(tyP1021McSetGen.tyNaviLyr1);
		IF p_tyNtParamCurr.tyDISettings.diMagWidthChkSen > 0 THEN
			tyP1021McSetGen.tyNaviLyr1.tyBitmapPageDisp.usiValueIdx := 3;
		ELSE
			tyP1021McSetGen.tyNaviLyr1.tyBitmapPageDisp.usiValueIdx := 1;
		END_IF

		fUIInRtStatOff(ADR(tyP1021McSetGen.tyGen.tyLyrGen1.uiRtStat));
		fUIInRtStatHide(ADR(tyP1021McSetGen.tyGen.tyLyrGen2.uiRtStat));
		fUIInRtStatHide(ADR(tyP1021McSetGen.tyGen.tyLyrGen3.uiRtStat));

		tyP1021McSetGen.tyNaviLyr3.tyBtnRgt.bRtCompl			:= FALSE;

	ELSIF tyP1021McSetGen.tyNaviLyr3.tyBtnLeft.bRtCompl = TRUE THEN
		p_tyC0004Navi ACCESS ADR(tyP1021McSetGen.tyNaviLyr2);
		IF p_tyNtParamCurr.tyDISettings.diMagWidthChkSen > 0 THEN
			tyP1021McSetGen.tyNaviLyr2.tyBitmapPageDisp.usiValueIdx := 4;
		ELSE
			tyP1021McSetGen.tyNaviLyr2.tyBitmapPageDisp.usiValueIdx := 2;
		END_IF

		fUIInRtStatHide(ADR(tyP1021McSetGen.tyGen.tyLyrGen1.uiRtStat));
		fUIInRtStatOff(ADR(tyP1021McSetGen.tyGen.tyLyrGen2.uiRtStat));
		fUIInRtStatHide(ADR(tyP1021McSetGen.tyGen.tyLyrGen3.uiRtStat));

		tyP1021McSetGen.tyNaviLyr3.tyBtnLeft.bRtCompl			:= FALSE;
	END_IF

END_ACTION
```

#### Act_OptP1021Teach.st
```iecst
ACTION Act_OptP1021Teach:

	IF tyP1021McSetGen.tyGen.tyBtnTravPosATeach.bRtCompl = TRUE THEN
		tyP1021McSetGen.tyGen.tyBtnTravPosATeach.bRtCompl	:= FALSE;
		tyP1021McSetGen.tyGen.tyBtnTravPosATeach.bValue		:= FALSE;

		bTeachTravPosA  	:= TRUE;
		eChgPage			:= UIP1026McSetTeach;

	ELSIF tyP1021McSetGen.tyGen.tyBtnTravPosBTeach.bRtCompl = TRUE THEN
		tyP1021McSetGen.tyGen.tyBtnTravPosBTeach.bRtCompl	:= FALSE;
		tyP1021McSetGen.tyGen.tyBtnTravPosBTeach.bValue		:= FALSE;

		bTeachTravPosB		:= TRUE;
		eChgPage			:= UIP1026McSetTeach;

	ELSIF tyP1021McSetGen.tyGen.tyBtnLiftPosATeach.bRtCompl = TRUE THEN
		tyP1021McSetGen.tyGen.tyBtnLiftPosATeach.bRtCompl	:= FALSE;
		tyP1021McSetGen.tyGen.tyBtnLiftPosATeach.bValue		:= FALSE;

		bTeachLifterPosA	:= TRUE;
		eChgPage			:= UIP1026McSetTeach;

	ELSIF tyP1021McSetGen.tyGen.tyBtnLiftPosBTeach.bRtCompl = TRUE THEN
		tyP1021McSetGen.tyGen.tyBtnLiftPosBTeach.bRtCompl	:= FALSE;
		tyP1021McSetGen.tyGen.tyBtnLiftPosBTeach.bValue		:= FALSE;

		bTeachLifterPosB	:= TRUE;
		eChgPage			:= UIP1026McSetTeach;

	END_IF

END_ACTION
```

#### Act_OptP1021Save.st
```iecst
ACTION Act_OptP1021Save:

	IF tyP1021McSetGen.tyGen.tyStringMcNm.bRtCompl					OR tyP1021McSetGen.tyGen.tyDrpDnDefaultMcMod.bRtCompl
		OR tyP1021McSetGen.tyGen.tyDrpDnDefaultFlippedBrd.bRtCompl	OR tyP1021McSetGen.tyGen.tyNumSSaverTm.bRtCompl
		OR tyP1021McSetGen.tyGen.tyBtnSSaverEn.bRtCompl				OR tyP1021McSetGen.tyGen.tyNumWidthAtHm.bRtCompl
		OR tyP1021McSetGen.tyGen.tyNumConvInitTm.bRtCompl			OR tyP1021McSetGen.tyGen.tyNumTranOutErrDlyTm.bRtCompl
		OR tyP1021McSetGen.tyGen.tyNumMag1ConvRunTm.bRtCompl		OR tyP1021McSetGen.tyGen.tyNumMag2ConvRunTm.bRtCompl
		OR tyP1021McSetGen.tyGen.tyNumMag3ConvRunTm.bRtCompl		OR tyP1021McSetGen.tyGen.tyNumMag4ConvRunTm.bRtCompl
		OR tyP1021McSetGen.tyGen.tyNumTravPosLaneA.bRtCompl
		OR tyP1021McSetGen.tyGen.tyNumLiftPosLaneA.bRtCompl			OR tyP1021McSetGen.tyGen.tyNumTravPosLaneB.bRtCompl
		OR tyP1021McSetGen.tyGen.tyNumLiftPosLaneB.bRtCompl			OR tyP1021McSetGen.tyGen.tyBtnAWDis.bRtCompl
		OR tyP1021McSetGen.tyGen.tyBtnMnlAccDat.bRtCompl			OR tyP1021McSetGen.tyGen.tyBtnAutoStepEn.bRtCompl
		OR tyP1021McSetGen.tyGen.tyBtnVSMEMAEn.bRtCompl				OR tyP1021McSetGen.tyGen.tyBtnHermesRmtEn.bRtCompl
		OR tyP1021McSetGen.tyGen.tyBtnLongBrdEn.bRtCompl			OR tyP1021McSetGen.tyGen.tyBtnOutShutterDis.bRtCompl
		OR tyP1021McSetGen.tyGen.tyBtnChgParamEn.bRtCompl			OR tyP1021McSetGen.tyGen.tyNumWidthOffset.bRtCompl
		OR tyP1021McSetGen.tyGen.tyNumMagAutoDetSenTm.bRtCompl		OR tyP1021McSetGen.tyGen.tyBtnAGVComEn.bRtCompl
		OR tyP1021McSetGen.tyGen.tyBtnLFBuzMute.bRtCompl			OR tyP1021McSetGen.tyGen.tyBtnAutoLogoutEn.bRtCompl
		OR tyP1021McSetGen.tyGen.tyNumAutoLogoutTm.bRtCompl			OR tyP1021McSetGen.tyGen.tyDrpDnAGVComProtocol.bRtCompl
		OR tyP1021McSetGen.tyGen.tyDrpDnMagExchangeMode.bRtCompl	OR tyP1021McSetGen.tyGen.tyBtnAGVSizeDisabled.bRtCompl
		OR tyP1021McSetGen.tyGen.tyBtnScannerEn.bRtCompl
		OR tyP1021McSetGen.tyGen.tyNumAWPusherAtHm.bRtCompl			OR tyP1021McSetGen.tyGen.tyBtnAWPusherDis.bRtCompl
		OR tyP1021McSetGen.tyGen.tyNumTravFixtoFixPosOutlet.bRtCompl
		OR tyP1021McSetGen.tyGen.tyBtnAWPusherDis.bRtCompl
		OR tyP1021McSetGen.tyGen.tyBtnDisableFMWarning.bRtCompl OR tyP1021McSetGen.tyGen.tyNumLMCFbTm.bRtCompl
		OR tyP1021McSetGen.tyGen.tyBtnMagWidthChkDis.bRtCompl	OR tyP1021McSetGen.tyGen.tyNumMag1WidthChkDetDist.bRtCompl
		OR tyP1021McSetGen.tyGen.tyNumMag2WidthChkDetDist.bRtCompl OR tyP1021McSetGen.tyGen.tyNumMag3WidthChkDetDist.bRtCompl
		OR tyP1021McSetGen.tyGen.tyBtnDBAOnRgtSen.bRtCompl OR tyP1021McSetGen.tyGen.tyBtnHermesSvyEn.bRtCompl     //new for Hermes 1.3
		OR tyP1021McSetGen.tyGen.tyBtnRFIDEn.bRtCompl OR tyP1021McSetGen.tyGen.tyNumRFIDWrTO.bRtCompl
		OR tyP1021McSetGen.tyGen.tyNumTravLaneBOffset.bRtCompl
		THEN

		fUIInRtStatHide(ADR(tyCommon.tySet.tyBtnSave.uiMaskRtStat));

		tyP1021McSetGen.tyGen.tyStringMcNm.bRtCompl				:= FALSE;
		tyP1021McSetGen.tyGen.tyDrpDnDefaultMcMod.bRtCompl		:= FALSE;
		tyP1021McSetGen.tyGen.tyDrpDnDefaultFlippedBrd.bRtCompl	:= FALSE;
		tyP1021McSetGen.tyGen.tyNumSSaverTm.bRtCompl			:= FALSE;
		tyP1021McSetGen.tyGen.tyBtnSSaverEn.bRtCompl			:= FALSE;
		tyP1021McSetGen.tyGen.tyNumWidthAtHm.bRtCompl			:= FALSE;
		tyP1021McSetGen.tyGen.tyNumConvInitTm.bRtCompl			:= FALSE;
		tyP1021McSetGen.tyGen.tyNumTranOutErrDlyTm.bRtCompl		:= FALSE;
		tyP1021McSetGen.tyGen.tyNumMag1ConvRunTm.bRtCompl		:= FALSE;
		tyP1021McSetGen.tyGen.tyNumMag2ConvRunTm.bRtCompl		:= FALSE;
		tyP1021McSetGen.tyGen.tyNumMag3ConvRunTm.bRtCompl 		:= FALSE;
		tyP1021McSetGen.tyGen.tyNumMag4ConvRunTm.bRtCompl 		:= FALSE;
		tyP1021McSetGen.tyGen.tyNumWidthOffset.bRtCompl			:= FALSE;
		tyP1021McSetGen.tyGen.tyNumMagAutoDetSenTm.bRtCompl		:= FALSE;
		tyP1021McSetGen.tyGen.tyBtnAGVComEn.bRtCompl			:= FALSE;
		tyP1021McSetGen.tyGen.tyBtnAutoLogoutEn.bRtCompl		:= FALSE;
		tyP1021McSetGen.tyGen.tyNumAutoLogoutTm.bRtCompl		:= FALSE;

		tyP1021McSetGen.tyGen.tyNumTravPosLaneA.bRtCompl		:= FALSE;
		tyP1021McSetGen.tyGen.tyNumLiftPosLaneA.bRtCompl		:= FALSE;
		tyP1021McSetGen.tyGen.tyNumTravPosLaneB.bRtCompl		:= FALSE;
		tyP1021McSetGen.tyGen.tyNumLiftPosLaneB.bRtCompl		:= FALSE;
		tyP1021McSetGen.tyGen.tyBtnAWDis.bRtCompl				:= FALSE;
		tyP1021McSetGen.tyGen.tyBtnMnlAccDat.bRtCompl			:= FALSE;
		tyP1021McSetGen.tyGen.tyBtnAutoStepEn.bRtCompl			:= FALSE;
		tyP1021McSetGen.tyGen.tyBtnVSMEMAEn.bRtCompl			:= FALSE;
		tyP1021McSetGen.tyGen.tyBtnHermesRmtEn.bRtCompl			:= FALSE;
		tyP1021McSetGen.tyGen.tyBtnLongBrdEn.bRtCompl			:= FALSE;
		tyP1021McSetGen.tyGen.tyBtnOutShutterDis.bRtCompl		:= FALSE;
		tyP1021McSetGen.tyGen.tyBtnChgParamEn.bRtCompl			:= FALSE;
		tyP1021McSetGen.tyGen.tyBtnLFBuzMute.bRtCompl			:= FALSE;
		tyP1021McSetGen.tyGen.tyDrpDnAGVComProtocol.bRtCompl	:= FALSE;
		tyP1021McSetGen.tyGen.tyDrpDnMagExchangeMode.bRtCompl	:= FALSE;
		tyP1021McSetGen.tyGen.tyBtnAGVSizeDisabled.bRtCompl		:= FALSE;
		tyP1021McSetGen.tyGen.tyBtnScannerEn.bRtCompl			:= FALSE;

		tyP1021McSetGen.tyGen.tyNumAWPusherAtHm.bRtCompl		:= FALSE;
		tyP1021McSetGen.tyGen.tyBtnAWPusherDis.bRtCompl			:= FALSE;
		tyP1021McSetGen.tyGen.tyNumTravFixtoFixPosOutlet.bRtCompl := FALSE;
		tyP1021McSetGen.tyGen.tyBtnDisableFMWarning.bRtCompl	:= FALSE;
		tyP1021McSetGen.tyGen.tyNumLMCFbTm.bRtCompl				:= FALSE;
		tyP1021McSetGen.tyGen.tyBtnMagWidthChkDis.bRtCompl		:= FALSE;
		tyP1021McSetGen.tyGen.tyNumMag1WidthChkDetDist.bRtCompl	:= FALSE;
		tyP1021McSetGen.tyGen.tyNumMag2WidthChkDetDist.bRtCompl	:= FALSE;
		tyP1021McSetGen.tyGen.tyNumMag3WidthChkDetDist.bRtCompl	:= FALSE;
		tyP1021McSetGen.tyGen.tyBtnDBAOnRgtSen.bRtCompl			:= FALSE;
		tyP1021McSetGen.tyGen.tyBtnHermesSvyEn.bRtCompl			:= FALSE; //new for Hermes 1.3
		tyP1021McSetGen.tyGen.tyBtnRFIDEn.bRtCompl 			:= FALSE;
		tyP1021McSetGen.tyGen.tyNumRFIDWrTO.bRtCompl 			:= FALSE;
		tyP1021McSetGen.tyGen.tyNumTravLaneBOffset.bRtCompl 	:= FALSE;

	END_IF

	IF tyCommon.tySet.tyBtnSave.bRtCompl = TRUE AND bSaveNetworkPriority=FALSE THEN

		tyMcParamWr.sMcNm					:=	tyP1021McSetGen.tyGen.tyStringMcNm.sValue;
		tyMcParamWr.usiDefaultMcMod			:=	tyP1021McSetGen.tyGen.tyDrpDnDefaultMcMod.usiValueIdx;
		tyMcParamWr.usiDefaultFlippedBrd	:=	tyP1021McSetGen.tyGen.tyDrpDnDefaultFlippedBrd.usiValueIdx;
		tyMcParamWr.uiSSaverTmInSec			:= 	DINT_TO_UINT(tyP1021McSetGen.tyGen.tyNumSSaverTm.diValue);
		tyMcParamWr.bSSaverEn				:=	tyP1021McSetGen.tyGen.tyBtnSSaverEn.bValue;
		tyMcParamWr.diWidthAtHmPosInUM		:=	tyP1021McSetGen.tyGen.tyNumWidthAtHm.diValue;
		tyMcParamWr.diConvInitTmInMS		:=	tyP1021McSetGen.tyGen.tyNumConvInitTm.diValue;
		tyMcParamWr.diTranOutErrDlyTmInMS	:=	tyP1021McSetGen.tyGen.tyNumTranOutErrDlyTm.diValue;
		tyMcParamWr.diMag1ConvRunTmOutInMS	:=	tyP1021McSetGen.tyGen.tyNumMag1ConvRunTm.diValue;
		tyMcParamWr.diMag2ConvRunTmOutInMS	:=	tyP1021McSetGen.tyGen.tyNumMag2ConvRunTm.diValue;
		tyMcParamWr.diMag3ConvRunTmOutInMS	:=	tyP1021McSetGen.tyGen.tyNumMag3ConvRunTm.diValue;
		tyMcParamWr.diMag4ConvRunTmOutInMS	:=	tyP1021McSetGen.tyGen.tyNumMag4ConvRunTm.diValue;
		tyMcParamWr.diWidthOffsetInUM		:=  tyP1021McSetGen.tyGen.tyNumWidthOffset.diValue;
		tyMcParamWr.diMagAutoDetectSenTmInMS:=  tyP1021McSetGen.tyGen.tyNumMagAutoDetSenTm.diValue;

		tyMcParamWr.diTravPosA				:=	tyP1021McSetGen.tyGen.tyNumTravPosLaneA.diValue;
		tyMcParamWr.diLifterPosA			:=	tyP1021McSetGen.tyGen.tyNumLiftPosLaneA.diValue;
		tyMcParamWr.diTravPosB				:=	tyP1021McSetGen.tyGen.tyNumTravPosLaneB.diValue;
		tyMcParamWr.diLifterPosB			:=	tyP1021McSetGen.tyGen.tyNumLiftPosLaneB.diValue;
		tyMcParamWr.bAWDis					:=	tyP1021McSetGen.tyGen.tyBtnAWDis.bValue;
		tyMcParamWr.bMnlAccDat				:=	tyP1021McSetGen.tyGen.tyBtnMnlAccDat.bValue;
		tyMcParamWr.bAutoStepEn				:=	tyP1021McSetGen.tyGen.tyBtnAutoStepEn.bValue;
		tyMcParamWr.bVSMEMAEn				:=	tyP1021McSetGen.tyGen.tyBtnVSMEMAEn.bValue;
		tyMcParamWr.bHermesRmtEn			:=	tyP1021McSetGen.tyGen.tyBtnHermesRmtEn.bValue;
		tyMcParamWr.bLongBrdEn				:=  tyP1021McSetGen.tyGen.tyBtnLongBrdEn.bValue;
		tyMcParamWr.bOutShutterDis			:=  tyP1021McSetGen.tyGen.tyBtnOutShutterDis.bValue;
		tyMcParamWr.bChgParamEn				:=  tyP1021McSetGen.tyGen.tyBtnChgParamEn.bValue;
		tyMcParamWr.bAGVComEn				:=  tyP1021McSetGen.tyGen.tyBtnAGVComEn.bValue;
		tyMcParamWr.bLFBuzMute				:=  tyP1021McSetGen.tyGen.tyBtnLFBuzMute.bValue;
		tyMcParamWr.bAutoLogoutEn			:=  tyP1021McSetGen.tyGen.tyBtnAutoLogoutEn.bValue;
		tyMcParamWr.diAutoLogoutTmInSec		:=  tyP1021McSetGen.tyGen.tyNumAutoLogoutTm.diValue;

		tyMcParamWr.eNetworkMod				:=  USINT_TO_DINT(tyP1021McSetGen.tyGen.tyDrpDnNetworkMod.usiValueIdx);
		tyMcParamWr.eAGVComProtocol			:=  tyP1021McSetGen.tyGen.tyDrpDnAGVComProtocol.usiValueIdx;
		tyMcParamWr.eMagExMode				:=  tyP1021McSetGen.tyGen.tyDrpDnMagExchangeMode.usiValueIdx;
		tyMcParamWr.bAIVSizeDisabled		:=  tyP1021McSetGen.tyGen.tyBtnAGVSizeDisabled.bValue;
		tyMcParamWr.bScannerEn				:=	tyP1021McSetGen.tyGen.tyBtnScannerEn.bValue;

		tyMcParamWr.diAWPusherAtHmPosInUM	:=	tyP1021McSetGen.tyGen.tyNumAWPusherAtHm.diValue;
		tyMcParamWr.bAWPusherDis			:=	tyP1021McSetGen.tyGen.tyBtnAWPusherDis.bValue;
		tyMcParamWr.diTravOutletFixtoFixPos	:=  tyP1021McSetGen.tyGen.tyNumTravFixtoFixPosOutlet.diValue;
		tyMcParamWr.bDisableFMWarning		:= 	tyP1021McSetGen.tyGen.tyBtnDisableFMWarning.bValue;
		tyMcParamWr.diLMCfbTmInMS 			:=	tyP1021McSetGen.tyGen.tyNumLMCFbTm.diValue;
		tyMcParamWr.bMagWidthChkDis 		:=	tyP1021McSetGen.tyGen.tyBtnMagWidthChkDis.bValue;
		tyMcParamWr.diMag1WidthChkDetDist 	:=  tyP1021McSetGen.tyGen.tyNumMag1WidthChkDetDist.diValue;
		tyMcParamWr.diMag2WidthChkDetDist 	:=  tyP1021McSetGen.tyGen.tyNumMag2WidthChkDetDist.diValue;
		tyMcParamWr.diMag3WidthChkDetDist 	:=  tyP1021McSetGen.tyGen.tyNumMag3WidthChkDetDist.diValue;
		tyMcParamWr.bDBAOnRgtSen			:=	tyP1021McSetGen.tyGen.tyBtnDBAOnRgtSen.bValue;
		tyMcParamWr.bHermesSvyEn			:= tyP1021McSetGen.tyGen.tyBtnHermesSvyEn.bValue;//new for Hermes 1.3
		tyMcParamWr.bMesRFIDEn				:= tyP1021McSetGen.tyGen.tyBtnRFIDEn.bValue;
		tyMcParamWr.diMesRFIDTOInMS			:= tyP1021McSetGen.tyGen.tyNumRFIDWrTO.diValue;
		tyMcParamWr.diTravLaneBOffset		:= tyP1021McSetGen.tyGen.tyNumTravLaneBOffset.diValue;

		IF tyP1021McSetGen.tyGen.tyDrpDnNetworkMod.usiValueIdx =DINT_TO_USINT(SetIPManually) THEN
			tyMcParamWr.sIPAddr				:= tyP1021McSetGen.tyGen.tyStringIPAddr.sValue;
			tyMcParamWr.sSubnetMask			:= tyP1021McSetGen.tyGen.tyStringSubnetMask.sValue;
		END_IF

		eMcParamAct	:= McParamActWrite;

		IF p_eMcParamStat = McParamActWrite AND p_eMcParamStatus = Done THEN
			eMcParamAct	:= McParamActIdle;

			usiNetworkModeOld := tyP1021McSetGen.tyGen.tyDrpDnNetworkMod.usiValueIdx;
			//Screen Saver Time
			tyProperty.tyVisu.uiSSaverTm	:= p_tyMcParamCurr.uiSSaverTmInSec;

			//Backup Param
			tyP1021McSetGen.tyGenBkUp	:= tyP1021McSetGen.tyGen;

			tyCommon.tySet.tyBtnSave.bRtCompl 	:= FALSE;
			fUIInRtStatOff(ADR(tyCommon.tySet.tyBtnSave.uiMaskRtStat));

		ELSIF p_eMcParamStatus = Error THEN
			p_tyC0008MsgBox ACCESS ADR(tyP1021McSetGen.tyMsgBoxSaveErr);

			IF tyP1021McSetGen.tyMsgBoxSaveErr.tyBtnNo.bRtCompl = TRUE THEN
				tyP1021McSetGen.tyMsgBoxSaveErr.tyBtnNo.bRtCompl	:= FALSE;
				tyP1021McSetGen.tyMsgBoxSaveErr.tyBtnNo.bValue		:= FALSE;

				p_tyC0008MsgBox ACCESS ADR(tyP1021McSetGen.tyMsgBoxHide);

				//Restore Param
				tyP1021McSetGen.tyGen	:= tyP1021McSetGen.tyGenBkUp;
				tyMcParamWr				:= p_tyMcParamCurr;

				tyCommon.tySet.tyBtnSave.bRtCompl 	:= FALSE;
				fUIInRtStatOff(ADR(tyCommon.tySet.tyBtnSave.uiMaskRtStat));

			END_IF

		END_IF

	END_IF

END_ACTION
```

#### Act_OptP1021Keypad.st
```iecst
ACTION Act_OptP1021Keypad:

	IF fUIOutRtStatTPIsOpen(ADR(tyP1021McSetGen.tyGen.tyStringMcNm.uiRtStat)) = TRUE THEN
		tyProperty.tyKeypad.tyStringTitle.sKeypadTitle	:= tyP1021McSetGen.tyGen.tyStringMcNm.sKeypadTitle;

	ELSIF fUIOutRtStatTPIsOpen(ADR(tyP1021McSetGen.tyGen.tyNumSSaverTm.uiRtStat)) = TRUE THEN
		tyProperty.tyKeypad.tyStringTitle.sKeypadTitle	:= tyP1021McSetGen.tyGen.tyNumSSaverTm.sKeypadTitle;

	ELSIF fUIOutRtStatTPIsOpen(ADR(tyP1021McSetGen.tyGen.tyStringIPAddr.uiRtStat)) = TRUE THEN
		tyProperty.tyKeypad.tyStringTitle.sKeypadTitle	:= tyP1021McSetGen.tyGen.tyStringIPAddr.sKeypadTitle;

	ELSIF fUIOutRtStatTPIsOpen(ADR(tyP1021McSetGen.tyGen.tyStringSubnetMask.uiRtStat)) = TRUE THEN
		tyProperty.tyKeypad.tyStringTitle.sKeypadTitle	:= tyP1021McSetGen.tyGen.tyStringSubnetMask.sKeypadTitle;

	ELSIF fUIOutRtStatTPIsOpen(ADR(tyP1021McSetGen.tyGen.tyNumConvInitTm.uiRtStat)) = TRUE THEN
		tyProperty.tyKeypad.tyStringTitle.sKeypadTitle	:= tyP1021McSetGen.tyGen.tyNumConvInitTm.sKeypadTitle;

	ELSIF fUIOutRtStatTPIsOpen(ADR(tyP1021McSetGen.tyGen.tyNumWidthAtHm.uiRtStat)) = TRUE THEN
		tyProperty.tyKeypad.tyStringTitle.sKeypadTitle	:= tyP1021McSetGen.tyGen.tyNumWidthAtHm.sKeypadTitle;

	ELSIF fUIOutRtStatTPIsOpen(ADR(tyP1021McSetGen.tyGen.tyNumTranOutErrDlyTm.uiRtStat)) = TRUE THEN
		tyProperty.tyKeypad.tyStringTitle.sKeypadTitle	:= tyP1021McSetGen.tyGen.tyNumTranOutErrDlyTm.sKeypadTitle;

	ELSIF fUIOutRtStatTPIsOpen(ADR(tyP1021McSetGen.tyGen.tyNumMag1ConvRunTm.uiRtStat)) = TRUE THEN
		tyProperty.tyKeypad.tyStringTitle.sKeypadTitle	:= tyP1021McSetGen.tyGen.tyNumMag1ConvRunTm.sKeypadTitle;

	ELSIF fUIOutRtStatTPIsOpen(ADR(tyP1021McSetGen.tyGen.tyNumMag2ConvRunTm.uiRtStat)) = TRUE THEN
		tyProperty.tyKeypad.tyStringTitle.sKeypadTitle	:= tyP1021McSetGen.tyGen.tyNumMag2ConvRunTm.sKeypadTitle;

	ELSIF fUIOutRtStatTPIsOpen(ADR(tyP1021McSetGen.tyGen.tyNumMag3ConvRunTm.uiRtStat)) = TRUE THEN
		tyProperty.tyKeypad.tyStringTitle.sKeypadTitle	:= tyP1021McSetGen.tyGen.tyNumMag3ConvRunTm.sKeypadTitle;

	ELSIF fUIOutRtStatTPIsOpen(ADR(tyP1021McSetGen.tyGen.tyNumMag4ConvRunTm.uiRtStat)) = TRUE THEN
		tyProperty.tyKeypad.tyStringTitle.sKeypadTitle	:= tyP1021McSetGen.tyGen.tyNumMag4ConvRunTm.sKeypadTitle;

	ELSIF fUIOutRtStatTPIsOpen(ADR(tyP1021McSetGen.tyGen.tyNumTravPosLaneA.uiRtStat)) = TRUE THEN
		tyProperty.tyKeypad.tyStringTitle.sKeypadTitle	:= tyP1021McSetGen.tyGen.tyNumTravPosLaneA.sKeypadTitle;

	ELSIF fUIOutRtStatTPIsOpen(ADR(tyP1021McSetGen.tyGen.tyNumTravPosLaneB.uiRtStat)) = TRUE THEN
		tyProperty.tyKeypad.tyStringTitle.sKeypadTitle	:= tyP1021McSetGen.tyGen.tyNumTravPosLaneB.sKeypadTitle;

	ELSIF fUIOutRtStatTPIsOpen(ADR(tyP1021McSetGen.tyGen.tyNumLiftPosLaneA.uiRtStat)) = TRUE THEN
		tyProperty.tyKeypad.tyStringTitle.sKeypadTitle	:= tyP1021McSetGen.tyGen.tyNumLiftPosLaneA.sKeypadTitle;

	ELSIF fUIOutRtStatTPIsOpen(ADR(tyP1021McSetGen.tyGen.tyNumLiftPosLaneB.uiRtStat)) = TRUE THEN
		tyProperty.tyKeypad.tyStringTitle.sKeypadTitle	:= tyP1021McSetGen.tyGen.tyNumLiftPosLaneB.sKeypadTitle;

	ELSIF fUIOutRtStatTPIsOpen(ADR(tyP1021McSetGen.tyGen.tyNumWidthOffset.uiRtStat)) = TRUE THEN
		tyProperty.tyKeypad.tyStringTitle.sKeypadTitle	:= tyP1021McSetGen.tyGen.tyNumWidthOffset.sKeypadTitle;

	ELSIF fUIOutRtStatTPIsOpen(ADR(tyP1021McSetGen.tyGen.tyNumMagAutoDetSenTm.uiRtStat)) = TRUE THEN
		tyProperty.tyKeypad.tyStringTitle.sKeypadTitle	:= tyP1021McSetGen.tyGen.tyNumMagAutoDetSenTm.sKeypadTitle;

	ELSIF fUIOutRtStatTPIsOpen(ADR(tyP1021McSetGen.tyNetwork.tyStringIPAddr.uiRtStat)) = TRUE THEN
		tyProperty.tyKeypad.tyStringTitle.sKeypadTitle	:= tyP1021McSetGen.tyNetwork.tyStringIPAddr.sKeypadTitle;

	ELSIF fUIOutRtStatTPIsOpen(ADR(tyP1021McSetGen.tyNetwork.tyStringSubnetMask.uiRtStat)) = TRUE THEN
		tyProperty.tyKeypad.tyStringTitle.sKeypadTitle	:= tyP1021McSetGen.tyNetwork.tyStringSubnetMask.sKeypadTitle;

	ELSIF fUIOutRtStatTPIsOpen(ADR(tyP1021McSetGen.tyGen.tyNumAWPusherAtHm.uiRtStat)) = TRUE THEN
		tyProperty.tyKeypad.tyStringTitle.sKeypadTitle	:= tyP1021McSetGen.tyGen.tyNumAWPusherAtHm.sKeypadTitle;

	ELSIF fUIOutRtStatTPIsOpen(ADR(tyP1021McSetGen.tyGen.tyNumLMCFbTm.uiRtStat)) = TRUE THEN
		tyProperty.tyKeypad.tyStringTitle.sKeypadTitle	:= tyP1021McSetGen.tyGen.tyNumLMCFbTm.sKeypadTitle;

	ELSIF fUIOutRtStatTPIsOpen(ADR(tyP1021McSetGen.tyGen.tyNumMag1WidthChkDetDist.uiRtStat)) = TRUE THEN
		tyProperty.tyKeypad.tyStringTitle.sKeypadTitle	:= tyP1021McSetGen.tyGen.tyNumMag1WidthChkDetDist.sKeypadTitle;
	ELSIF fUIOutRtStatTPIsOpen(ADR(tyP1021McSetGen.tyGen.tyNumMag2WidthChkDetDist.uiRtStat)) = TRUE THEN
		tyProperty.tyKeypad.tyStringTitle.sKeypadTitle	:= tyP1021McSetGen.tyGen.tyNumMag2WidthChkDetDist.sKeypadTitle;
	ELSIF fUIOutRtStatTPIsOpen(ADR(tyP1021McSetGen.tyGen.tyNumMag3WidthChkDetDist.uiRtStat)) = TRUE THEN
		tyProperty.tyKeypad.tyStringTitle.sKeypadTitle	:= tyP1021McSetGen.tyGen.tyNumMag3WidthChkDetDist.sKeypadTitle;

	ELSE
		tyProperty.tyKeypad.tyStringTitle.sKeypadTitle	:= '';

	END_IF

END_ACTION
```

#### Act_OptP1024Save.st
```iecst
ACTION Act_OptP1024Save:

	IF tyP1024McSetAntiGap.tyAntiGap.tyNumLftSenOff.bRtCompl
		OR tyP1024McSetAntiGap.tyAntiGap.tyNumRgtSenOff.bRtCompl
		OR tyP1024McSetAntiGap.tyAntiGap.tyNumMagConvEntOn.bRtCompl
		OR tyP1024McSetAntiGap.tyAntiGap.tyNumMagConvEntOff.bRtCompl
		OR tyP1024McSetAntiGap.tyAntiGap.tyNumMagConvPresentOn.bRtCompl
		OR tyP1024McSetAntiGap.tyAntiGap.tyNumMagConvPresentOff.bRtCompl
		THEN

		fUIInRtStatHide(ADR(tyCommon.tySet.tyBtnSave.uiMaskRtStat));

		tyP1024McSetAntiGap.tyAntiGap.tyNumLftSenOff.bRtCompl	:= FALSE;
		tyP1024McSetAntiGap.tyAntiGap.tyNumRgtSenOff.bRtCompl	:= FALSE;
		tyP1024McSetAntiGap.tyAntiGap.tyNumMagConvEntOn.bRtCompl	:= FALSE;
		tyP1024McSetAntiGap.tyAntiGap.tyNumMagConvEntOff.bRtCompl	:= FALSE;
		tyP1024McSetAntiGap.tyAntiGap.tyNumMagConvPresentOn.bRtCompl	:= FALSE;
		tyP1024McSetAntiGap.tyAntiGap.tyNumMagConvPresentOff.bRtCompl	:= FALSE;
	END_IF

	IF tyCommon.tySet.tyBtnSave.bRtCompl = TRUE THEN

		tyMcParamWr.tyLftSenAntiGapDly.diSigOffTm	:=  tyP1024McSetAntiGap.tyAntiGap.tyNumLftSenOff.diValue;
		tyMcParamWr.tyRgtSenAntiGapDly.diSigOffTm	:=	tyP1024McSetAntiGap.tyAntiGap.tyNumRgtSenOff.diValue;
		tyMcParamWr.tyMagConvEntrySenAntiGapDly.diSigOnTm	:=  tyP1024McSetAntiGap.tyAntiGap.tyNumMagConvEntOn.diValue;
		tyMcParamWr.tyMagConvEntrySenAntiGapDly.diSigOffTm	:=  tyP1024McSetAntiGap.tyAntiGap.tyNumMagConvEntOff.diValue;
		tyMcParamWr.tyMagConvPresentSenAntiGapDly.diSigOnTm	:=	tyP1024McSetAntiGap.tyAntiGap.tyNumMagConvPresentOn.diValue;
		tyMcParamWr.tyMagConvPresentSenAntiGapDly.diSigOffTm:=	tyP1024McSetAntiGap.tyAntiGap.tyNumMagConvPresentOff.diValue;

		eMcParamAct	:= McParamActWrite;

		IF p_eMcParamStat = McParamActWrite AND p_eMcParamStatus = Done THEN

			eMcParamAct	:= McParamActIdle;

			//Update BackUp Param
			tyP1024McSetAntiGap.tyAntiGapBkUp	:= tyP1024McSetAntiGap.tyAntiGap;

			tyCommon.tySet.tyBtnSave.bRtCompl 	:= FALSE;
			fUIInRtStatOff(ADR(tyCommon.tySet.tyBtnSave.uiMaskRtStat));

		ELSIF p_eMcParamStatus = Error THEN
			p_tyC0008MsgBox ACCESS ADR(tyP1024McSetAntiGap.tyMsgBoxSaveErr);

			IF tyP1024McSetAntiGap.tyMsgBoxSaveErr.tyBtnNo.bRtCompl = TRUE THEN
				tyP1024McSetAntiGap.tyMsgBoxSaveErr.tyBtnNo.bRtCompl	:= FALSE;
				tyP1024McSetAntiGap.tyMsgBoxSaveErr.tyBtnNo.bValue		:= FALSE;

				p_tyC0008MsgBox ACCESS ADR(tyP1024McSetAntiGap.tyMsgBoxHide);

				//Restore Param
				tyP1024McSetAntiGap.tyAntiGap	:= tyP1024McSetAntiGap.tyAntiGapBkUp;
				tyMcParamWr						:= p_tyMcParamCurr;

				tyCommon.tySet.tyBtnSave.bRtCompl 	:= FALSE;
				fUIInRtStatOff(ADR(tyCommon.tySet.tyBtnSave.uiMaskRtStat));
			END_IF

		END_IF

	END_IF

END_ACTION
```

#### Act_EntP1022Disp.st
```iecst
ACTION Act_EntP1022Disp:
	//Access Address
	//new for Hermes 1.3
	IF p_tyNtParamCurr.bLFPrep OR p_tyNtParamCurr.bLCSLFPrep OR p_tyNtParamCurr.bLCSReqRcpPrep OR p_tyNtParamCurr.bLCSManageRcpPrep OR p_tyNtParamCurr.bLCSLiveDatPrep
		OR p_tyNtParamCurr.bLFUsrSetPrep OR p_tyNtParamCurr.bLFUsrSetPrep (*OR  p_tyNtParamCurr.bUSWidthChkPrep*) OR p_tyNtParamCurr.bDSWidthChkPrep THEN
		bNaviLyr1 := TRUE;
	ELSE
		bNaviLyr1 := FALSE;
	END_IF

	IF (p_tyNtParamCurr.bHermesSvyPrep AND p_tyMcParamCurr.bHermesSvyEn)  THEN
		bNaviLyr2 := TRUE;
	ELSE
		bNaviLyr2 := FALSE;
	END_IF

	//Access Address
	IF bNaviLyr1 AND NOT bNaviLyr2 THEN
		p_tyC0004Navi ACCESS ADR(tyP1022McSetVComm.tyNaviLyr1);
		fUIInRtStatOff(ADR(tyP1022McSetVComm.tyVComSel.tyLyr.uiRtStat)); //show
		fUIInRtStatHide(ADR(tyP1022McSetVComm.tyVComSvy.tyLyr.uiRtStat));
		fUIInRtStatOff(ADR(tyP1022McSetVComm.tyLF.tyLyr.uiRtStat)); //show

	ELSIF NOT bNaviLyr1 AND bNaviLyr2 THEN
		p_tyC0004Navi ACCESS ADR(tyP1022McSetVComm.tyNaviLyr2);
		fUIInRtStatHide(ADR(tyP1022McSetVComm.tyVComSel.tyLyr.uiRtStat)); //show
		fUIInRtStatOff(ADR(tyP1022McSetVComm.tyVComSvy.tyLyr.uiRtStat));
		fUIInRtStatHide(ADR(tyP1022McSetVComm.tyLF.tyLyr.uiRtStat)); //show

	ELSIF bNaviLyr1 AND bNaviLyr2 THEN
		p_tyC0004Navi ACCESS ADR(tyP1022McSetVComm.tyNaviLyr3);
		fUIInRtStatOff(ADR(tyP1022McSetVComm.tyVComSel.tyLyr.uiRtStat)); //show
		fUIInRtStatHide(ADR(tyP1022McSetVComm.tyVComSvy.tyLyr.uiRtStat));
		fUIInRtStatOff(ADR(tyP1022McSetVComm.tyLF.tyLyr.uiRtStat)); //show
	END_IF
	//p_tyC0004Navi ACCESS ADR(tyP1022McSetVComm.tyNaviBack);

	p_tyC0005Main ACCESS ADR(tyCommon.tyMain);

	p_tyC0006Set ACCESS ADR(tyCommon.tySet);

	p_tyC0007Notif ACCESS ADR(tyCommon.tyNotif);

	p_tyC0008MsgBox ACCESS ADR(tyP1022McSetVComm.tyMsgBoxHide);

	p_tyC0009Info ACCESS ADR(tyCommon.tyInfo);

	p_tyP1022McSetVCommSel ACCESS ADR(tyP1022McSetVComm.tyVComSel);
	p_tyP1022McSetVCommLF ACCESS ADR(tyP1022McSetVComm.tyLF);
	p_tyP1022McSetVCommSvy ACCESS ADR(tyP1022McSetVComm.tyVComSvy); //new for Hermes 1.3

	//Backup Param
	tyP1022McSetVComm.tyVComSelBkUp	:= tyP1022McSetVComm.tyVComSel;
	tyP1022McSetVComm.tyLFBkUp		:= tyP1022McSetVComm.tyLF;
	tyP1022McSetVComm.tyVComSvyBkUp	:= tyP1022McSetVComm.tyVComSvy; //new for Hermes 1.3

END_ACTION
```

#### Act_ExitP1022.st
```iecst
ACTION Act_ExitP1022:

	IF tyCommon.tySet.tyBtnSave.uiMaskRtStat.0 = FALSE THEN
		usiChgPage	:= 1;

	ELSE

		p_tyC0008MsgBox ACCESS ADR(tyP1022McSetVComm.tyMsgBoxExitAsk);

		IF tyP1022McSetVComm.tyMsgBoxExitAsk.tyBtnYes.bRtCompl = TRUE THEN
			tyP1022McSetVComm.tyMsgBoxExitAsk.tyBtnYes.bRtCompl	:= FALSE;
			tyP1022McSetVComm.tyMsgBoxExitAsk.tyBtnYes.bValue	:= FALSE;

			p_tyC0008MsgBox ACCESS ADR(tyP1022McSetVComm.tyMsgBoxHide);

			//Restore Param
			tyP1022McSetVComm.tyVComSel	:= tyP1022McSetVComm.tyVComSelBkUp;
			tyP1022McSetVComm.tyLF		:= tyP1022McSetVComm.tyLFBkUp;
			tyP1022McSetVComm.tyVComSvy	:= tyP1022McSetVComm.tyVComSvyBkUp; //new for Hermes 1.3

			fUIInRtStatOff(ADR(tyCommon.tySet.tyBtnSave.uiMaskRtStat));

			usiChgPage	:= 1;

		ELSIF tyP1022McSetVComm.tyMsgBoxExitAsk.tyBtnNo.bRtCompl = TRUE THEN
			tyP1022McSetVComm.tyMsgBoxExitAsk.tyBtnNo.bRtCompl	:= FALSE;
			tyP1022McSetVComm.tyMsgBoxExitAsk.tyBtnNo.bValue	:= FALSE;

			p_tyC0008MsgBox ACCESS ADR(tyP1022McSetVComm.tyMsgBoxHide);

			eChgPage	:= eCurrPage;
			usiChgPage	:= 0;

		END_IF

	END_IF

END_ACTION
```

#### Act_OptP1022Keypad.st
```iecst
ACTION Act_OptP1022Keypad:

	IF fUIOutRtStatTPIsOpen(ADR(tyP1022McSetVComm.tyVComSvy.tyNumSndAliveTm.uiRtStat)) = TRUE THEN
		tyProperty.tyKeypad.tyStringTitle.sKeypadTitle	:= tyP1022McSetVComm.tyVComSvy.tyNumSndAliveTm.sKeypadTitle;

	ELSIF fUIOutRtStatTPIsOpen(ADR(tyP1022McSetVComm.tyVComSvy.tyNumSvySystemPort.uiRtStat)) = TRUE THEN
		tyProperty.tyKeypad.tyStringTitle.sKeypadTitle	:= tyP1022McSetVComm.tyVComSvy.tyNumSvySystemPort.sKeypadTitle;

	END_IF

END_ACTION
```

#### Act_OptP1022Navi.st
```iecst
ACTION Act_OptP1022Navi:

	tyP1022McSetVComm.tyNaviBack.tyBtnBack.bRtLk	:= tyCommon.tySet.tyBtnSave.bRtCompl;

	IF tyP1022McSetVComm.tyNaviLyr1.tyBtnBack.bRtCompl OR tyP1022McSetVComm.tyNaviLyr2.tyBtnBack.bRtCompl OR
		tyP1022McSetVComm.tyNaviLyr3.tyBtnBack.bRtCompl OR tyP1022McSetVComm.tyNaviLyr4.tyBtnBack.bRtCompl THEN
		tyP1022McSetVComm.tyNaviLyr1.tyBtnBack.bRtCompl	:= FALSE;
		tyP1022McSetVComm.tyNaviLyr2.tyBtnBack.bRtCompl	:= FALSE;
		tyP1022McSetVComm.tyNaviLyr3.tyBtnBack.bRtCompl	:= FALSE;
		tyP1022McSetVComm.tyNaviLyr4.tyBtnBack.bRtCompl	:= FALSE;

		eChgPage	:= UIP1020McSetNavi;

	ELSIF tyP1022McSetVComm.tyNaviLyr3.tyBtnLeft.bRtCompl = TRUE OR tyP1022McSetVComm.tyNaviLyr3.tyBtnRgt.bRtCompl = TRUE THEN
		tyP1022McSetVComm.tyNaviLyr3.tyBtnLeft.bRtCompl	:= FALSE;
		tyP1022McSetVComm.tyNaviLyr3.tyBtnRgt.bRtCompl	:= FALSE;

		p_tyC0004Navi ACCESS ADR(tyP1022McSetVComm.tyNaviLyr4);

		fUIInRtStatHide(ADR(tyP1022McSetVComm.tyVComSel.tyLyr.uiRtStat));
		fUIInRtStatOff(ADR(tyP1022McSetVComm.tyVComSvy.tyLyr.uiRtStat)); //new for Hermes 1.3
		fUIInRtStatHide(ADR(tyP1022McSetVComm.tyLF.tyLyr.uiRtStat));

	ELSIF tyP1022McSetVComm.tyNaviLyr4.tyBtnLeft.bRtCompl = TRUE OR tyP1022McSetVComm.tyNaviLyr4.tyBtnRgt.bRtCompl = TRUE THEN
		tyP1022McSetVComm.tyNaviLyr4.tyBtnLeft.bRtCompl	:= FALSE;
		tyP1022McSetVComm.tyNaviLyr4.tyBtnRgt.bRtCompl	:= FALSE;

		p_tyC0004Navi ACCESS ADR(tyP1022McSetVComm.tyNaviLyr3);

		fUIInRtStatOff(ADR(tyP1022McSetVComm.tyVComSel.tyLyr.uiRtStat));
		fUIInRtStatHide(ADR(tyP1022McSetVComm.tyVComSvy.tyLyr.uiRtStat));  //new for Hermes 1.3
		fUIInRtStatOff(ADR(tyP1022McSetVComm.tyLF.tyLyr.uiRtStat));
	END_IF

END_ACTION
```

#### Act_OptP1022Save.st
```iecst
ACTION Act_OptP1022Save:

	IF tyP1022McSetVComm.tyVComSel.tyBtnLF.bRtCompl 			OR tyP1022McSetVComm.tyVComSel.tyBtnLCSLF.bRtCompl
		OR tyP1022McSetVComm.tyVComSel.tyBtnLCSReqRcp.bRtCompl	OR tyP1022McSetVComm.tyVComSel.tyBtnLCSManageRcp.bRtCompl
		OR tyP1022McSetVComm.tyVComSel.tyBtnLCSLiveDat.bRtCompl	OR tyP1022McSetVComm.tyLF.tyBtnLeaderMc.bRtCompl
		OR tyP1022McSetVComm.tyLF.tyBtnSectionLdr.bRtCompl		OR tyP1022McSetVComm.tyLF.tyBtnDSWidthChkEn.bRtCompl
		OR tyP1022McSetVComm.tyLF.tyBtnDBAOnWOAlign.bRtCompl
		OR tyP1022McSetVComm.tyVComSvy.tyBtnConfiguration.bRtCompl //new for Hermes 1.3
		OR tyP1022McSetVComm.tyVComSvy.tyBtnCheckAliveResponse.bRtCompl OR tyP1022McSetVComm.tyVComSvy.tyBtnBoardTracking.bRtCompl //new for Hermes 1.3
		OR tyP1022McSetVComm.tyVComSvy.tyBtnQueryWorkOrderInfo.bRtCompl OR tyP1022McSetVComm.tyVComSvy.tyBtnSendWorkOrderInfo.bRtCompl //new for Hermes 1.3
		OR tyP1022McSetVComm.tyVComSvy.tyNumSndAliveTm.bRtCompl         OR tyP1022McSetVComm.tyVComSvy.tyNumSvySystemPort.bRtCompl	   //new for Hermes 1.3
		THEN
		fUIInRtStatHide(ADR(tyCommon.tySet.tyBtnSave.uiMaskRtStat));

		IF (NOT p_tyNtParamCurr.bLFUsrSetPrep AND NOT p_tyNtParamCurr.bLeaderMc) OR (p_tyNtParamCurr.bLFUsrSetPrep AND NOT tyP1022McSetVComm.tyLF.tyBtnLeaderMc.bValue) THEN
			IF tyP1022McSetVComm.tyVComSel.tyBtnLF.bRtCompl AND tyP1022McSetVComm.tyVComSel.tyBtnLF.bValue THEN
				tyP1022McSetVComm.tyVComSel.tyBtnLCSLF.bValue	:= FALSE;
			ELSIF tyP1022McSetVComm.tyVComSel.tyBtnLCSLF.bRtCompl AND tyP1022McSetVComm.tyVComSel.tyBtnLCSLF.bValue THEN
				tyP1022McSetVComm.tyVComSel.tyBtnLF.bValue		:= FALSE;
			END_IF

			IF tyP1022McSetVComm.tyVComSel.tyBtnLF.bValue = TRUE AND tyP1022McSetVComm.tyVComSel.tyBtnLCSLF.bValue = TRUE THEN
				tyP1022McSetVComm.tyVComSel.tyBtnLF.bValue		:= FALSE;
				tyP1022McSetVComm.tyVComSel.tyBtnLCSLF.bValue	:= FALSE;
			END_IF
		END_IF

		tyP1022McSetVComm.tyVComSel.tyBtnLF.bRtCompl			:= FALSE;
		tyP1022McSetVComm.tyVComSel.tyBtnLCSLF.bRtCompl			:= FALSE;
		tyP1022McSetVComm.tyVComSel.tyBtnLCSReqRcp.bRtCompl		:= FALSE;
		tyP1022McSetVComm.tyVComSel.tyBtnLCSManageRcp.bRtCompl	:= FALSE;
		tyP1022McSetVComm.tyVComSel.tyBtnLCSLiveDat.bRtCompl	:= FALSE;

		tyP1022McSetVComm.tyLF.tyBtnLeaderMc.bRtCompl			:= FALSE;
		tyP1022McSetVComm.tyLF.tyBtnSectionLdr.bRtCompl			:= FALSE;
		tyP1022McSetVComm.tyLF.tyBtnDSWidthChkEn.bRtCompl		:= FALSE;
		tyP1022McSetVComm.tyLF.tyBtnDBAOnWOAlign.bRtCompl		:= FALSE;

		//new for Hermes 1.3
		tyP1022McSetVComm.tyVComSvy.tyBtnConfiguration.bRtCompl			:= FALSE;
		tyP1022McSetVComm.tyVComSvy.tyBtnCheckAliveResponse.bRtCompl	:= FALSE;
		tyP1022McSetVComm.tyVComSvy.tyBtnBoardTracking.bRtCompl			:= FALSE;
		tyP1022McSetVComm.tyVComSvy.tyBtnQueryWorkOrderInfo.bRtCompl	:= FALSE;
		tyP1022McSetVComm.tyVComSvy.tyBtnSendWorkOrderInfo.bRtCompl		:= FALSE;
		tyP1022McSetVComm.tyVComSvy.tyNumSndAliveTm.bRtCompl			:= FALSE;
		tyP1022McSetVComm.tyVComSvy.tyNumSvySystemPort.bRtCompl			:= FALSE;
	END_IF

	IF tyCommon.tySet.tyBtnSave.bRtCompl = TRUE THEN

		tyMcParamWr.bLFEn			:=  tyP1022McSetVComm.tyVComSel.tyBtnLF.bValue;
		tyMcParamWr.bLCSLFEn		:=  tyP1022McSetVComm.tyVComSel.tyBtnLCSLF.bValue;
		tyMcParamWr.bLCSReqRcpEn	:=  tyP1022McSetVComm.tyVComSel.tyBtnLCSReqRcp.bValue;
		tyMcParamWr.bLCSManageRcpEn	:=  tyP1022McSetVComm.tyVComSel.tyBtnLCSManageRcp.bValue;
		tyMcParamWr.bLCSLiveDatEn	:=  tyP1022McSetVComm.tyVComSel.tyBtnLCSLiveDat.bValue;

		tyMcParamWr.bLFLeaderMc		:=	tyP1022McSetVComm.tyLF.tyBtnLeaderMc.bValue;
		tyMcParamWr.bSectionLeader	:=	tyP1022McSetVComm.tyLF.tyBtnSectionLdr.bValue;
		tyMcParamWr.bDSWidthChkEn	:= 	tyP1022McSetVComm.tyLF.tyBtnDSWidthChkEn.bValue;
		tyMcParamWr.bDBAOnWOAlign	:= 	tyP1022McSetVComm.tyLF.tyBtnDBAOnWOAlign.bValue;

		//new for Hermes 1.3
		tyHermesSvyParamWr.bFeatureConfiguration	    	:=	tyP1022McSetVComm.tyVComSvy.tyBtnConfiguration.bValue;
		tyHermesSvyParamWr.bFeatureCheckAliveResponse		:=	tyP1022McSetVComm.tyVComSvy.tyBtnCheckAliveResponse.bValue;
		tyHermesSvyParamWr.bFeatureBoardTracking	    	:=	tyP1022McSetVComm.tyVComSvy.tyBtnBoardTracking.bValue;
		tyHermesSvyParamWr.bFeatureQueryWorkOrderInfo		:=	tyP1022McSetVComm.tyVComSvy.tyBtnQueryWorkOrderInfo.bValue;
		tyHermesSvyParamWr.bFeatureSendWorkOrderInfo		:=	tyP1022McSetVComm.tyVComSvy.tyBtnSendWorkOrderInfo.bValue;
		tyHermesSvyParamWr.tSndAlive		                :=	DINT_TO_TIME(tyP1022McSetVComm.tyVComSvy.tyNumSndAliveTm.diValue);
		tyHermesSvyParamWr.uiSvySvstemPort		            :=	DINT_TO_UINT(tyP1022McSetVComm.tyVComSvy.tyNumSvySystemPort.diValue);
		bSaveHMISvyConfig := TRUE;

		eMcParamAct	:= McParamActWrite;
		eHermesAct	:= HermesActWriteConfig; //new for Hermes 1.3

		IF p_eMcParamStat = McParamActWrite AND p_eMcParamStatus = Done THEN
			eMcParamAct	:= McParamActIdle;
			eHermesAct	:= HermesActIdle;  //new for Hermes 1.3

			//Update BackUp Param
			tyP1022McSetVComm.tyVComSelBkUp	:= tyP1022McSetVComm.tyVComSel;
			tyP1022McSetVComm.tyLFBkUp		:= tyP1022McSetVComm.tyLF;
			tyP1022McSetVComm.tyVComSvyBkUp	:= tyP1022McSetVComm.tyVComSvy;  //new for Hermes 1.3

			tyCommon.tySet.tyBtnSave.bRtCompl	:= FALSE;
			fUIInRtStatOff(ADR(tyCommon.tySet.tyBtnSave.uiMaskRtStat));
			bSaveHMISvyConfig := FALSE;  //new for Hermes 1.3

		ELSIF p_eMcParamStatus = Error THEN
			p_tyC0008MsgBox ACCESS ADR(tyP1022McSetVComm.tyMsgBoxSaveErr);

			IF tyP1022McSetVComm.tyMsgBoxSaveErr.tyBtnNo.bRtCompl = TRUE THEN
				tyP1022McSetVComm.tyMsgBoxSaveErr.tyBtnNo.bRtCompl 	:= FALSE;
				tyP1022McSetVComm.tyMsgBoxSaveErr.tyBtnNo.bValue	:= FALSE;

				p_tyC0008MsgBox ACCESS ADR(tyP1022McSetVComm.tyMsgBoxHide);

				//Restore Param
				tyP1022McSetVComm.tyVComSel	:= tyP1022McSetVComm.tyVComSelBkUp;
				tyP1022McSetVComm.tyVComSvy	:= tyP1022McSetVComm.tyVComSvyBkUp;  //new for Hermes 1.3
				tyP1022McSetVComm.tyLF		:= tyP1022McSetVComm.tyLFBkUp;
				tyMcParamWr					:= p_tyMcParamCurr;
				bSaveHMISvyConfig := FALSE;  //new for Hermes 1.3

				tyCommon.tySet.tyBtnSave.bRtCompl 	:= FALSE;
				fUIInRtStatOff(ADR(tyCommon.tySet.tyBtnSave.uiMaskRtStat));

			END_IF

		END_IF

	END_IF

END_ACTION
```

#### Act_EntP1023Disp.st
```iecst
ACTION Act_EntP1023Disp:

	//Access Address
	IF p_tyNtParamCurr.bProjLaneBPrep THEN
		p_tyC0004Navi ACCESS ADR(tyP1023McSetHComm.tyNaviLyr1);
	ELSE
		p_tyC0004Navi ACCESS ADR(tyP1023McSetHComm.tyNaviBack);
	END_IF

	p_tyC0005Main ACCESS ADR(tyCommon.tyMain);

	p_tyC0006Set ACCESS ADR(tyCommon.tySet);

	p_tyC0007Notif ACCESS ADR(tyCommon.tyNotif);

	p_tyC0008MsgBox ACCESS ADR(tyP1023McSetHComm.tyMsgBoxHide);

	p_tyC0009Info ACCESS ADR(tyCommon.tyInfo);

	p_tyP1023McSetHCommDSSel ACCESS ADR(tyP1023McSetHComm.tyDSSelA);
	p_tyP1023McSetHCommDSSMEMA ACCESS ADR(tyP1023McSetHComm.tyDSSMEMAA);
	p_tyP1023McSetHCommDSHermes ACCESS ADR(tyP1023McSetHComm.tyDSHermesA);

	//Backup Param
	tyP1023McSetHComm.tyDSSelABkUp		:= tyP1023McSetHComm.tyDSSelA;
	tyP1023McSetHComm.tyDSSMEMAABkUp	:= tyP1023McSetHComm.tyDSSMEMAA;
	tyP1023McSetHComm.tyDSHermesABkUp	:= tyP1023McSetHComm.tyDSHermesA;
	tyP1023McSetHComm.tyDSSelBBkUp		:= tyP1023McSetHComm.tyDSSelB;
	tyP1023McSetHComm.tyDSSMEMABBkUp	:= tyP1023McSetHComm.tyDSSMEMAB;
	tyP1023McSetHComm.tyDSHermesBBkUp	:= tyP1023McSetHComm.tyDSHermesB;

END_ACTION
```

#### Act_ExitP1023.st
```iecst
ACTION Act_ExitP1023:

	IF tyCommon.tySet.tyBtnSave.uiMaskRtStat.0 = FALSE THEN
		usiChgPage	:= 1;

	ELSE

		p_tyC0008MsgBox ACCESS ADR(tyP1023McSetHComm.tyMsgBoxExitAsk);

		IF tyP1023McSetHComm.tyMsgBoxExitAsk.tyBtnYes.bRtCompl = TRUE THEN
			tyP1023McSetHComm.tyMsgBoxExitAsk.tyBtnYes.bRtCompl	:= FALSE;
			tyP1023McSetHComm.tyMsgBoxExitAsk.tyBtnYes.bValue	:= FALSE;

			p_tyC0008MsgBox ACCESS ADR(tyP1023McSetHComm.tyMsgBoxHide);

			//Restore Param
			tyP1023McSetHComm.tyDSSelA		:= tyP1023McSetHComm.tyDSSelABkUp;
			tyP1023McSetHComm.tyDSSMEMAA	:= tyP1023McSetHComm.tyDSSMEMAABkUp;
			tyP1023McSetHComm.tyDSHermesA	:= tyP1023McSetHComm.tyDSHermesABkUp;

			tyP1023McSetHComm.tyDSSelB		:= tyP1023McSetHComm.tyDSSelBBkUp;
			tyP1023McSetHComm.tyDSSMEMAB	:= tyP1023McSetHComm.tyDSSMEMABBkUp;
			tyP1023McSetHComm.tyDSHermesB	:= tyP1023McSetHComm.tyDSHermesBBkUp;

			fUIInRtStatOff(ADR(tyCommon.tySet.tyBtnSave.uiMaskRtStat));

			usiChgPage	:= 1;

		ELSIF tyP1023McSetHComm.tyMsgBoxExitAsk.tyBtnNo.bRtCompl = TRUE THEN
			tyP1023McSetHComm.tyMsgBoxExitAsk.tyBtnNo.bRtCompl	:= FALSE;
			tyP1023McSetHComm.tyMsgBoxExitAsk.tyBtnNo.bValue	:= FALSE;

			p_tyC0008MsgBox ACCESS ADR(tyP1023McSetHComm.tyMsgBoxHide);

			eChgPage	:= eCurrPage;
			usiChgPage	:= 0;

		END_IF

	END_IF

END_ACTION
```

#### Act_OptP1023Navi.st
```iecst
ACTION Act_OptP1023Navi:

	tyP1023McSetHComm.tyNaviBack.tyBtnBack.bRtLk	:= tyCommon.tySet.tyBtnSave.bRtCompl;
	tyP1023McSetHComm.tyNaviLyr1.tyBtnBack.bRtLk	:= tyCommon.tySet.tyBtnSave.bRtCompl;
	tyP1023McSetHComm.tyNaviLyr2.tyBtnBack.bRtLk	:= tyCommon.tySet.tyBtnSave.bRtCompl;

	IF tyP1023McSetHComm.tyNaviLyr1.tyBtnBack.bRtCompl = TRUE OR tyP1023McSetHComm.tyNaviLyr2.tyBtnBack.bRtCompl = TRUE OR tyP1023McSetHComm.tyNaviBack.tyBtnBack.bRtCompl = TRUE THEN
		eChgPage	:= UIP1020McSetNavi;

		tyP1023McSetHComm.tyNaviLyr1.tyBtnBack.bRtCompl		:= FALSE;
		tyP1023McSetHComm.tyNaviLyr2.tyBtnBack.bRtCompl		:= FALSE;
		tyP1023McSetHComm.tyNaviBack.tyBtnBack.bRtCompl		:= FALSE;

	ELSIF tyP1023McSetHComm.tyNaviLyr1.tyBtnLeft.bRtCompl = TRUE OR tyP1023McSetHComm.tyNaviLyr1.tyBtnRgt.bRtCompl = TRUE THEN

		p_tyC0004Navi ACCESS ADR(tyP1023McSetHComm.tyNaviLyr2);
		p_tyP1023McSetHCommDSSel ACCESS ADR(tyP1023McSetHComm.tyDSSelB);
		p_tyP1023McSetHCommDSSMEMA ACCESS ADR(tyP1023McSetHComm.tyDSSMEMAB);
		p_tyP1023McSetHCommDSHermes ACCESS ADR(tyP1023McSetHComm.tyDSHermesB);

		tyP1023McSetHComm.tyDSSelB.tyBtnHermes.uiRtStat.0	:= NOT p_tyNtParamCurr.bHermesPrep;

		tyP1023McSetHComm.tyNaviLyr1.tyBtnLeft.bRtCompl	:= FALSE;
		tyP1023McSetHComm.tyNaviLyr1.tyBtnRgt.bRtCompl	:= FALSE;

	ELSIF tyP1023McSetHComm.tyNaviLyr2.tyBtnLeft.bRtCompl = TRUE OR tyP1023McSetHComm.tyNaviLyr2.tyBtnRgt.bRtCompl = TRUE THEN

		p_tyC0004Navi ACCESS ADR(tyP1023McSetHComm.tyNaviLyr1);
		p_tyP1023McSetHCommDSSel ACCESS ADR(tyP1023McSetHComm.tyDSSelA);
		p_tyP1023McSetHCommDSSMEMA ACCESS ADR(tyP1023McSetHComm.tyDSSMEMAA);
		p_tyP1023McSetHCommDSHermes ACCESS ADR(tyP1023McSetHComm.tyDSHermesA);

		tyP1023McSetHComm.tyDSSelA.tyBtnHermes.uiRtStat.0	:= NOT p_tyNtParamCurr.bHermesPrep;

		tyP1023McSetHComm.tyNaviLyr2.tyBtnLeft.bRtCompl	:= FALSE;
		tyP1023McSetHComm.tyNaviLyr2.tyBtnRgt.bRtCompl	:= FALSE;

	END_IF

END_ACTION
```

#### Act_OptP1023ShowLyr.st
```iecst
ACTION Act_OptP1023ShowLyr:

	//Downstream A
	IF tyP1023McSetHComm.tyDSSelA.tyLyr.uiRtStat.0 = FALSE THEN

		IF tyP1023McSetHComm.tyDSSelA.tyBtnSMEMA.bValue = TRUE THEN

			fUIInRtStatOff(ADR(tyP1023McSetHComm.tyDSSMEMAA.tyLyr.uiRtStat));
			fUIInRtStatHide(ADR(tyP1023McSetHComm.tyDSHermesA.tyLyr.uiRtStat));

			tyP1023McSetHComm.tyDSSMEMAA.tyBtnGdSig.uiRtStat.0	:= NOT(tyP1023McSetHComm.tyDSSMEMAA.tyDrpDnSMEMAMod.usiValueIdx = 2);

		ELSIF tyP1023McSetHComm.tyDSSelA.tyBtnHermes.bValue = TRUE THEN

			fUIInRtStatHide(ADR(tyP1023McSetHComm.tyDSSMEMAA.tyLyr.uiRtStat));
			fUIInRtStatOff(ADR(tyP1023McSetHComm.tyDSHermesA.tyLyr.uiRtStat));

			//Mask
			tyP1023McSetHComm.tyDSHermesA.tyBitmapMask.uiMaskRtStat.0	:= NOT((p_tyNtParamCurr.bHermesRmtPrep = TRUE AND p_tyMcParamCurr.bHermesRmtEn = TRUE) OR (p_tyNtParamCurr.bHermesSvyPrep = TRUE AND p_tyMcParamCurr.bHermesSvyEn = TRUE)); //new for Hermes 1.3 //True = Hide, False = Show
		END_IF

	ELSE

		fUIInRtStatHide(ADR(tyP1023McSetHComm.tyDSSMEMAA.tyLyr.uiRtStat));
		fUIInRtStatHide(ADR(tyP1023McSetHComm.tyDSHermesA.tyLyr.uiRtStat));

	END_IF

	//Downstream B
	IF tyP1023McSetHComm.tyDSSelB.tyLyr.uiRtStat.0 = FALSE THEN

		IF tyP1023McSetHComm.tyDSSelB.tyBtnSMEMA.bValue = TRUE THEN

			fUIInRtStatOff(ADR(tyP1023McSetHComm.tyDSSMEMAB.tyLyr.uiRtStat));
			fUIInRtStatHide(ADR(tyP1023McSetHComm.tyDSHermesB.tyLyr.uiRtStat));

			tyP1023McSetHComm.tyDSSMEMAB.tyBtnGdSig.uiRtStat.0	:= NOT(tyP1023McSetHComm.tyDSSMEMAB.tyDrpDnSMEMAMod.usiValueIdx = 2);

		ELSIF tyP1023McSetHComm.tyDSSelB.tyBtnHermes.bValue = TRUE THEN

			fUIInRtStatHide(ADR(tyP1023McSetHComm.tyDSSMEMAB.tyLyr.uiRtStat));
			fUIInRtStatOff(ADR(tyP1023McSetHComm.tyDSHermesB.tyLyr.uiRtStat));

			//Mask
			tyP1023McSetHComm.tyDSHermesB.tyBitmapMask.uiMaskRtStat.0	:= NOT((p_tyNtParamCurr.bHermesRmtPrep = TRUE AND p_tyMcParamCurr.bHermesRmtEn = TRUE) OR (p_tyNtParamCurr.bHermesSvyPrep = TRUE AND p_tyMcParamCurr.bHermesSvyEn = TRUE)); //new for Hermes 1.3 //True = Hide, False = Show
		END_IF

	ELSE

		fUIInRtStatHide(ADR(tyP1023McSetHComm.tyDSSMEMAB.tyLyr.uiRtStat));
		fUIInRtStatHide(ADR(tyP1023McSetHComm.tyDSHermesB.tyLyr.uiRtStat));

	END_IF

END_ACTION
```

#### Act_OptP1023Save.st
```iecst
ACTION Act_OptP1023Save:

	IF tyP1023McSetHComm.tyDSSelA.tyBtnSMEMA.bRtCompl				OR tyP1023McSetHComm.tyDSSelA.tyBtnHermes.bRtCompl
		OR tyP1023McSetHComm.tyDSSMEMAA.tyDrpDnSMEMAMod.bRtCompl	OR tyP1023McSetHComm.tyDSSMEMAA.tyBtnGdSig.bRtCompl
		OR tyP1023McSetHComm.tyDSHermesA.tyNumSndAliveTm.bRtCompl	OR tyP1023McSetHComm.tyDSHermesA.tyNumLaneID.bRtCompl
		OR tyP1023McSetHComm.tyDSHermesA.tyNumSvrPort.bRtCompl		OR tyP1023McSetHComm.tyDSHermesA.tyBtnCheckAliveResponse.bRtCompl
		OR tyP1023McSetHComm.tyDSHermesA.tyBtnBoardForecast.bRtCompl	OR tyP1023McSetHComm.tyDSHermesA.tyBtnSendBoardInfo.bRtCompl

		OR tyP1023McSetHComm.tyDSSelB.tyBtnSMEMA.bRtCompl			OR tyP1023McSetHComm.tyDSSelB.tyBtnHermes.bRtCompl
		OR tyP1023McSetHComm.tyDSSMEMAB.tyDrpDnSMEMAMod.bRtCompl	OR tyP1023McSetHComm.tyDSSMEMAB.tyBtnGdSig.bRtCompl
		OR tyP1023McSetHComm.tyDSHermesB.tyNumSndAliveTm.bRtCompl	OR tyP1023McSetHComm.tyDSHermesB.tyNumLaneID.bRtCompl
		OR tyP1023McSetHComm.tyDSHermesB.tyNumSvrPort.bRtCompl		OR tyP1023McSetHComm.tyDSHermesB.tyBtnCheckAliveResponse.bRtCompl
		OR tyP1023McSetHComm.tyDSHermesB.tyBtnBoardForecast.bRtCompl	OR tyP1023McSetHComm.tyDSHermesB.tyBtnSendBoardInfo.bRtCompl THEN

		fUIInRtStatHide(ADR(tyCommon.tySet.tyBtnSave.uiMaskRtStat));

		tyP1023McSetHComm.tyDSSMEMAA.tyDrpDnSMEMAMod.bRtCompl			:= FALSE;
		tyP1023McSetHComm.tyDSSMEMAA.tyBtnGdSig.bRtCompl				:= FALSE;
		tyP1023McSetHComm.tyDSHermesA.tyNumSndAliveTm.bRtCompl			:= FALSE;
		tyP1023McSetHComm.tyDSHermesA.tyNumLaneID.bRtCompl				:= FALSE;
		tyP1023McSetHComm.tyDSHermesA.tyNumSvrPort.bRtCompl				:= FALSE;
		tyP1023McSetHComm.tyDSHermesA.tyBtnCheckAliveResponse.bRtCompl	:= FALSE;
		tyP1023McSetHComm.tyDSHermesA.tyBtnBoardForecast.bRtCompl		:= FALSE;
		tyP1023McSetHComm.tyDSHermesA.tyBtnSendBoardInfo.bRtCompl		:= FALSE;

		tyP1023McSetHComm.tyDSSMEMAB.tyDrpDnSMEMAMod.bRtCompl			:= FALSE;
		tyP1023McSetHComm.tyDSSMEMAB.tyBtnGdSig.bRtCompl				:= FALSE;
		tyP1023McSetHComm.tyDSHermesB.tyNumSndAliveTm.bRtCompl			:= FALSE;
		tyP1023McSetHComm.tyDSHermesB.tyNumLaneID.bRtCompl				:= FALSE;
		tyP1023McSetHComm.tyDSHermesB.tyNumSvrPort.bRtCompl				:= FALSE;
		tyP1023McSetHComm.tyDSHermesB.tyBtnCheckAliveResponse.bRtCompl	:= FALSE;
		tyP1023McSetHComm.tyDSHermesB.tyBtnBoardForecast.bRtCompl		:= FALSE;
		tyP1023McSetHComm.tyDSHermesB.tyBtnSendBoardInfo.bRtCompl		:= FALSE;
	END_IF

	//new for Hermes 1.3
	//Auto de-select
//	IF EDGEPOS(tyP1023McSetHComm.tyUSHermes.tyBtnCmpTypeId.bValue) THEN
//		tyP1023McSetHComm.tyUSHermes.tyBtnOverWrite.bValue := FALSE;
//	ELSIF EDGEPOS(tyP1023McSetHComm.tyUSHermes.tyBtnCmpParam.bValue) THEN
//		tyP1023McSetHComm.tyUSHermes.tyBtnCmpTypeId.bValue := TRUE;
//	ELSIF EDGEPOS(tyP1023McSetHComm.tyUSHermes.tyBtnCmpTypeId.bValue = FALSE) THEN
//		tyP1023McSetHComm.tyUSHermes.tyBtnCmpParam.bValue := FALSE;
//	ELSIF EDGEPOS(tyP1023McSetHComm.tyUSHermes.tyBtnOverWrite.bValue = TRUE) THEN
//		tyP1023McSetHComm.tyUSHermes.tyBtnCmpTypeId.bValue := FALSE;
//	END_IF
	bSaveHMIConfigure := tyCommon.tySet.tyBtnSave.bRtCompl;

	IF tyCommon.tySet.tyBtnSave.bRtCompl = TRUE THEN

		IF usiSaveCommStep = 0 THEN
			//Save Machine Parameter
			//Downstream A
			IF tyP1023McSetHComm.tyDSSelA.tyBtnSMEMA.bValue = TRUE THEN
				tyMcParamWr.eDSCommA	:= McSetCommModSMEMA;
			ELSIF tyP1023McSetHComm.tyDSSelA.tyBtnHermes.bValue = TRUE THEN
				tyMcParamWr.eDSCommA	:= McSetCommModHermes;
			END_IF

			tyMcParamWr.tyDSCommASMEMA.eSelection		:= USINT_TO_UDINT(tyP1023McSetHComm.tyDSSMEMAA.tyDrpDnSMEMAMod.usiValueIdx);
			tyMcParamWr.tyDSCommASMEMA.bStatSigSetGd	:= tyP1023McSetHComm.tyDSSMEMAA.tyBtnGdSig.bValue;

			//Downstream B
			IF tyP1023McSetHComm.tyDSSelB.tyBtnSMEMA.bValue = TRUE THEN
				tyMcParamWr.eDSCommB	:= McSetCommModSMEMA;
			ELSIF tyP1023McSetHComm.tyDSSelB.tyBtnHermes.bValue = TRUE THEN
				tyMcParamWr.eDSCommB	:= McSetCommModHermes;
			END_IF

			tyMcParamWr.tyDSCommBSMEMA.eSelection		:= USINT_TO_UDINT(tyP1023McSetHComm.tyDSSMEMAB.tyDrpDnSMEMAMod.usiValueIdx);
			tyMcParamWr.tyDSCommBSMEMA.bStatSigSetGd	:= tyP1023McSetHComm.tyDSSMEMAB.tyBtnGdSig.bValue;

			eMcParamAct	:= McParamActWrite;

			IF p_eMcParamStat = McParamActWrite AND p_eMcParamStatus = Done THEN
				eMcParamAct	:= McParamActIdle;

				//Update BackUp Param
				tyP1023McSetHComm.tyDSSelABkUp 		:= tyP1023McSetHComm.tyDSSelA;
				tyP1023McSetHComm.tyDSSMEMAABkUp	:= tyP1023McSetHComm.tyDSSMEMAA;
				tyP1023McSetHComm.tyDSSelBBkUp		:= tyP1023McSetHComm.tyDSSelB;
				tyP1023McSetHComm.tyDSSMEMABBkUp	:= tyP1023McSetHComm.tyDSSMEMAB;

				usiSaveCommStep	:= 1;

				bHCommModChg := TRUE; // to opsmag1,2,3
			ELSIF p_eMcParamStatus = Error THEN
				p_tyC0008MsgBox ACCESS ADR(tyP1023McSetHComm.tyMsgBoxSaveErr);

				IF tyP1023McSetHComm.tyMsgBoxSaveErr.tyBtnNo.bRtCompl = TRUE THEN
					tyP1023McSetHComm.tyMsgBoxSaveErr.tyBtnNo.bRtCompl	:= FALSE;
					tyP1023McSetHComm.tyMsgBoxSaveErr.tyBtnNo.bValue	:= FALSE;

					p_tyC0008MsgBox ACCESS ADR(tyP1023McSetHComm.tyMsgBoxHide);

					//Restore Param
					tyP1023McSetHComm.tyDSSelA		:= tyP1023McSetHComm.tyDSSelABkUp;
					tyP1023McSetHComm.tyDSSMEMAA	:= tyP1023McSetHComm.tyDSSMEMAABkUp;
					tyP1023McSetHComm.tyDSSelB		:= tyP1023McSetHComm.tyDSSelBBkUp;
					tyP1023McSetHComm.tyDSSMEMAB	:= tyP1023McSetHComm.tyDSSMEMABBkUp;

					tyMcParamWr	:= p_tyMcParamCurr;

					usiSaveCommStep	:= 1;
				END_IF

			END_IF

		ELSIF usiSaveCommStep = 1 THEN
			//Save Hermes Configuration
			//Downstream A
			a_tyHermesDSParamWr[0].tSndAlive					:= DINT_TO_TIME(tyP1023McSetHComm.tyDSHermesA.tyNumSndAliveTm.diValue);
			a_tyHermesDSParamWr[0].uiSvrPort					:= DINT_TO_UINT(tyP1023McSetHComm.tyDSHermesA.tyNumSvrPort.diValue);
			a_tyHermesDSParamWr[0].iLaneID						:= DINT_TO_INT(tyP1023McSetHComm.tyDSHermesA.tyNumLaneID.diValue);
			a_tyHermesDSParamWr[0].bFeatureCheckAliveResponse	:= tyP1023McSetHComm.tyDSHermesA.tyBtnCheckAliveResponse.bValue;
			a_tyHermesDSParamWr[0].bFeatureBoardForecast	    := tyP1023McSetHComm.tyDSHermesA.tyBtnBoardForecast.bValue;
			a_tyHermesDSParamWr[0].bFeatureSendBoardInfo    	:= tyP1023McSetHComm.tyDSHermesA.tyBtnSendBoardInfo.bValue;

			//Downstream B
			a_tyHermesDSParamWr[1].tSndAlive					:= DINT_TO_TIME(tyP1023McSetHComm.tyDSHermesB.tyNumSndAliveTm.diValue);
			a_tyHermesDSParamWr[1].uiSvrPort					:= DINT_TO_UINT(tyP1023McSetHComm.tyDSHermesB.tyNumSvrPort.diValue);
			a_tyHermesDSParamWr[1].iLaneID						:= DINT_TO_INT(tyP1023McSetHComm.tyDSHermesB.tyNumLaneID.diValue);
			a_tyHermesDSParamWr[1].bFeatureCheckAliveResponse	:= tyP1023McSetHComm.tyDSHermesB.tyBtnCheckAliveResponse.bValue;
			a_tyHermesDSParamWr[1].bFeatureBoardForecast	    := tyP1023McSetHComm.tyDSHermesB.tyBtnBoardForecast.bValue;
			a_tyHermesDSParamWr[1].bFeatureSendBoardInfo    	:= tyP1023McSetHComm.tyDSHermesB.tyBtnSendBoardInfo.bValue;

			eHermesAct	:= HermesActWriteConfig;

			IF p_eHermesStat = HermesActWriteConfig AND p_eHermesStatus = Done THEN
				eHermesAct	:= HermesActIdle;

				//Update BackUp Param
				tyP1023McSetHComm.tyDSHermesABkUp	:= tyP1023McSetHComm.tyDSHermesA;
				tyP1023McSetHComm.tyDSHermesBBkUp	:= tyP1023McSetHComm.tyDSHermesB;

				usiSaveCommStep	:= 0;

				tyCommon.tySet.tyBtnSave.bRtCompl	:= FALSE;

				fUIInRtStatOff(ADR(tyCommon.tySet.tyBtnSave.uiMaskRtStat));

			ELSIF p_eMcParamStatus = Error THEN
				p_tyC0008MsgBox ACCESS ADR(tyP1023McSetHComm.tyMsgBoxSaveErr);

				IF tyP1023McSetHComm.tyMsgBoxSaveErr.tyBtnNo.bRtCompl = TRUE THEN
					tyP1023McSetHComm.tyMsgBoxSaveErr.tyBtnNo.bRtCompl	:= FALSE;
					tyP1023McSetHComm.tyMsgBoxSaveErr.tyBtnNo.bValue	:= FALSE;

					p_tyC0008MsgBox ACCESS ADR(tyP1023McSetHComm.tyMsgBoxHide);

					//Restore Param
					tyP1023McSetHComm.tyDSHermesA	:= tyP1023McSetHComm.tyDSHermesABkUp;
					tyP1023McSetHComm.tyDSHermesB	:= tyP1023McSetHComm.tyDSHermesBBkUp;

					a_tyHermesDSParamWr				:= p_tyHermesConfiguration.a_tyDSParam;

					tyCommon.tySet.tyBtnSave.bRtCompl 	:= FALSE;

					fUIInRtStatOff(ADR(tyCommon.tySet.tyBtnSave.uiMaskRtStat));

					usiSaveCommStep	:= 0;
				END_IF

			END_IF

		ELSIF usiSaveCommStep = 99 THEN
			//Message: IP Address Invalid
			p_tyC0008MsgBox ACCESS ADR(tyP1023McSetHComm.tyMsgBoxIPAddrInvalid);

			IF tyP1023McSetHComm.tyMsgBoxIPAddrInvalid.tyBtnNo.bRtCompl = TRUE THEN
				tyP1023McSetHComm.tyMsgBoxIPAddrInvalid.tyBtnNo.bRtCompl	:= FALSE;
				tyP1023McSetHComm.tyMsgBoxIPAddrInvalid.tyBtnNo.bValue		:= FALSE;

				p_tyC0008MsgBox ACCESS ADR(tyP1023McSetHComm.tyMsgBoxHide);

				//Restore Param
				tyP1023McSetHComm.tyDSSelA		:= tyP1023McSetHComm.tyDSSelABkUp;
				tyP1023McSetHComm.tyDSSMEMAA	:= tyP1023McSetHComm.tyDSSMEMAABkUp;
				tyP1023McSetHComm.tyDSHermesA	:= tyP1023McSetHComm.tyDSHermesABkUp;
				tyP1023McSetHComm.tyDSSelB		:= tyP1023McSetHComm.tyDSSelBBkUp;
				tyP1023McSetHComm.tyDSSMEMAB	:= tyP1023McSetHComm.tyDSSMEMABBkUp;
				tyP1023McSetHComm.tyDSHermesB	:= tyP1023McSetHComm.tyDSHermesBBkUp;

				tyCommon.tySet.tyBtnSave.bRtCompl 	:= FALSE;

				fUIInRtStatOff(ADR(tyCommon.tySet.tyBtnSave.uiMaskRtStat));

				usiSaveCommStep	:= 0;
			END_IF

		END_IF

	END_IF

END_ACTION
```

#### Act_OptP1023USSel.st
```iecst
ACTION Act_OptP1023USSel:

	IF tyP1023McSetHComm.tyUSSel.tyBtnSMEMA.bRtCompl = TRUE THEN
		tyP1023McSetHComm.tyUSSel.tyBtnSMEMA.bRtCompl	:= FALSE;

		tyP1023McSetHComm.tyUSSel.tyBtnSMEMA.bValue		:= TRUE;
		tyP1023McSetHComm.tyUSSel.tyBtnSMEMA.bRtLk		:= TRUE;

		tyP1023McSetHComm.tyUSSel.tyBtnHermes.bValue	:= FALSE;
		tyP1023McSetHComm.tyUSSel.tyBtnHermes.bRtLk		:= FALSE;

	ELSIF tyP1023McSetHComm.tyUSSel.tyBtnHermes.bRtCompl = TRUE THEN
		tyP1023McSetHComm.tyUSSel.tyBtnHermes.bRtCompl	:= FALSE;

		tyP1023McSetHComm.tyUSSel.tyBtnSMEMA.bValue		:= FALSE;
		tyP1023McSetHComm.tyUSSel.tyBtnSMEMA.bRtLk		:= FALSE;

		tyP1023McSetHComm.tyUSSel.tyBtnHermes.bValue	:= TRUE;
		tyP1023McSetHComm.tyUSSel.tyBtnHermes.bRtLk		:= TRUE;

	END_IF

END_ACTION
```

#### Act_OptP1023DSSel.st
```iecst
ACTION Act_OptP1023DSSel:

	//Select SMEMA Communication A
	IF tyP1023McSetHComm.tyDSSelA.tyBtnSMEMA.bRtCompl = TRUE THEN
		tyP1023McSetHComm.tyDSSelA.tyBtnSMEMA.bRtCompl	:= FALSE;

		tyP1023McSetHComm.tyDSSelA.tyBtnSMEMA.bValue	:= TRUE;
		tyP1023McSetHComm.tyDSSelA.tyBtnSMEMA.bRtLk		:= TRUE;

		tyP1023McSetHComm.tyDSSelA.tyBtnHermes.bValue	:= FALSE;
		tyP1023McSetHComm.tyDSSelA.tyBtnHermes.bRtLk	:= FALSE;

	//Select Hermes Communication A
	ELSIF tyP1023McSetHComm.tyDSSelA.tyBtnHermes.bRtCompl = TRUE THEN
		tyP1023McSetHComm.tyDSSelA.tyBtnHermes.bRtCompl	:= FALSE;

		tyP1023McSetHComm.tyDSSelA.tyBtnSMEMA.bValue	:= FALSE;
		tyP1023McSetHComm.tyDSSelA.tyBtnSMEMA.bRtLk		:= FALSE;

		tyP1023McSetHComm.tyDSSelA.tyBtnHermes.bValue	:= TRUE;
		tyP1023McSetHComm.tyDSSelA.tyBtnHermes.bRtLk	:= TRUE;

	END_IF

	//Select SMEMA Communication B
	IF tyP1023McSetHComm.tyDSSelB.tyBtnSMEMA.bRtCompl = TRUE THEN
		tyP1023McSetHComm.tyDSSelB.tyBtnSMEMA.bRtCompl	:= FALSE;

		tyP1023McSetHComm.tyDSSelB.tyBtnSMEMA.bValue	:= TRUE;
		tyP1023McSetHComm.tyDSSelB.tyBtnSMEMA.bRtLk		:= TRUE;

		tyP1023McSetHComm.tyDSSelB.tyBtnHermes.bValue	:= FALSE;
		tyP1023McSetHComm.tyDSSelB.tyBtnHermes.bRtLk	:= FALSE;

		//Select Hermes Communication B
	ELSIF tyP1023McSetHComm.tyDSSelB.tyBtnHermes.bRtCompl = TRUE THEN
		tyP1023McSetHComm.tyDSSelB.tyBtnHermes.bRtCompl	:= FALSE;

		tyP1023McSetHComm.tyDSSelB.tyBtnSMEMA.bValue	:= FALSE;
		tyP1023McSetHComm.tyDSSelB.tyBtnSMEMA.bRtLk		:= FALSE;

		tyP1023McSetHComm.tyDSSelB.tyBtnHermes.bValue	:= TRUE;
		tyP1023McSetHComm.tyDSSelB.tyBtnHermes.bRtLk	:= TRUE;

	END_IF

END_ACTION
```

#### Act_OptP1023Keypad.st
```iecst
ACTION Act_OptP1023Keypad:

	//Downstream A
	IF fUIOutRtStatTPIsOpen(ADR(tyP1023McSetHComm.tyDSHermesA.tyNumSndAliveTm.uiRtStat)) = TRUE THEN
		tyProperty.tyKeypad.tyStringTitle.sKeypadTitle	:= tyP1023McSetHComm.tyDSHermesA.tyNumSndAliveTm.sKeypadTitle;

	ELSIF fUIOutRtStatTPIsOpen(ADR(tyP1023McSetHComm.tyDSHermesA.tyNumLaneID.uiRtStat)) = TRUE THEN
		tyProperty.tyKeypad.tyStringTitle.sKeypadTitle	:= tyP1023McSetHComm.tyDSHermesA.tyNumLaneID.sKeypadTitle;

	ELSIF fUIOutRtStatTPIsOpen(ADR(tyP1023McSetHComm.tyDSHermesA.tyNumSvrPort.uiRtStat)) = TRUE THEN
		tyProperty.tyKeypad.tyStringTitle.sKeypadTitle	:= tyP1023McSetHComm.tyDSHermesA.tyNumSvrPort.sKeypadTitle;

	END_IF

	//Downstream B
	IF fUIOutRtStatTPIsOpen(ADR(tyP1023McSetHComm.tyDSHermesB.tyNumSndAliveTm.uiRtStat)) = TRUE THEN
		tyProperty.tyKeypad.tyStringTitle.sKeypadTitle	:= tyP1023McSetHComm.tyDSHermesB.tyNumSndAliveTm.sKeypadTitle;

	ELSIF fUIOutRtStatTPIsOpen(ADR(tyP1023McSetHComm.tyDSHermesB.tyNumLaneID.uiRtStat)) = TRUE THEN
		tyProperty.tyKeypad.tyStringTitle.sKeypadTitle	:= tyP1023McSetHComm.tyDSHermesB.tyNumLaneID.sKeypadTitle;

	ELSIF fUIOutRtStatTPIsOpen(ADR(tyP1023McSetHComm.tyDSHermesB.tyNumSvrPort.uiRtStat)) = TRUE THEN
		tyProperty.tyKeypad.tyStringTitle.sKeypadTitle	:= tyP1023McSetHComm.tyDSHermesB.tyNumSvrPort.sKeypadTitle;

	END_IF

END_ACTION
```

#### Act_EntP1025Disp.st
```iecst
ACTION Act_EntP1025Disp:

	//Access Address
	p_tyC0004Navi ACCESS ADR(tyP1025McSetAIVComm.tyNaviBack);

	p_tyC0005Main ACCESS ADR(tyCommon.tyMain);

	p_tyC0006Set ACCESS ADR(tyCommon.tySet);

	p_tyC0007Notif ACCESS ADR(tyCommon.tyNotif);

	p_tyC0008MsgBox ACCESS ADR (tyP1025McSetAIVComm.tyMsgBoxHide);

	p_tyC0009Info ACCESS ADR(tyCommon.tyInfo);

	p_tyP1025McSetAIVComm ACCESS ADR(tyP1025McSetAIVComm.tyAIVComm);

	//Backup Param
	tyP1025McSetAIVComm.tyAIVCommBkUp	:= tyP1025McSetAIVComm.tyAIVComm;

END_ACTION
```

#### Act_ExitP1025.st
```iecst
ACTION Act_ExitP1025:

	IF tyCommon.tySet.tyBtnSave.uiMaskRtStat.0 = FALSE THEN
		usiChgPage	:= 1;

	ELSE

		p_tyC0008MsgBox ACCESS ADR(tyP1025McSetAIVComm.tyMsgBoxExitAsk);

		IF tyP1025McSetAIVComm.tyMsgBoxExitAsk.tyBtnYes.bRtCompl = TRUE THEN
			tyP1025McSetAIVComm.tyMsgBoxExitAsk.tyBtnYes.bRtCompl	:= FALSE;
			tyP1025McSetAIVComm.tyMsgBoxExitAsk.tyBtnYes.bValue		:= FALSE;

			p_tyC0008MsgBox ACCESS ADR(tyP1025McSetAIVComm.tyMsgBoxHide);

			//Restore Param
			tyP1025McSetAIVComm.tyAIVComm	:= tyP1025McSetAIVComm.tyAIVCommBkUp;

			fUIInRtStatOff(ADR(tyCommon.tySet.tyBtnSave.uiMaskRtStat));

			usiChgPage	:= 1;

		ELSIF tyP1025McSetAIVComm.tyMsgBoxExitAsk.tyBtnNo.bRtCompl = TRUE THEN
			tyP1025McSetAIVComm.tyMsgBoxExitAsk.tyBtnNo.bRtCompl	:= FALSE;
			tyP1025McSetAIVComm.tyMsgBoxExitAsk.tyBtnNo.bValue		:= FALSE;

			p_tyC0008MsgBox ACCESS ADR(tyP1025McSetAIVComm.tyMsgBoxHide);

			eChgPage	:= eCurrPage;
			usiChgPage	:= 0;

		END_IF

	END_IF

END_ACTION
```

#### Act_OptP1025Keypad.st
```iecst
ACTION Act_OptP1025Keypad:

	IF fUIOutRtStatTPIsOpen(ADR(tyP1025McSetAIVComm.tyAIVComm.tyNumSvrPort.uiRtStat)) = TRUE THEN
		tyProperty.tyKeypad.tyStringTitle.sKeypadTitle	:= tyP1025McSetAIVComm.tyAIVComm.tyNumSvrPort.sKeypadTitle;

	ELSIF fUIOutRtStatTPIsOpen(ADR(tyP1025McSetAIVComm.tyAIVComm.tyNumAllwClntPort.uiRtStat)) = TRUE THEN
		tyProperty.tyKeypad.tyStringTitle.sKeypadTitle	:= tyP1025McSetAIVComm.tyAIVComm.tyNumAllwClntPort.sKeypadTitle;

	ELSIF fUIOutRtStatTPIsOpen(ADR(tyP1025McSetAIVComm.tyAIVComm.tyStringAllwClntIP.uiRtStat)) = TRUE THEN
		tyProperty.tyKeypad.tyStringTitle.sKeypadTitle	:= tyP1025McSetAIVComm.tyAIVComm.tyStringAllwClntIP.sKeypadTitle;

	END_IF

END_ACTION
```

#### Act_OptP1025Navi.st
```iecst
ACTION Act_OptP1025Navi:

	tyP1025McSetAIVComm.tyNaviBack.tyBtnBack.bRtLk	:= tyCommon.tySet.tyBtnSave.bRtCompl;

	IF tyP1025McSetAIVComm.tyNaviBack.tyBtnBack.bRtCompl = TRUE THEN
		tyP1025McSetAIVComm.tyNaviBack.tyBtnBack.bRtCompl	:= FALSE;

		eChgPage	:= UIP1020McSetNavi;

	END_IF

END_ACTION
```
